LIN {X 0,Y 221.844,Z 433.494,A -85,B 0,C 180,E1 -25932.083,E2 -25932.083} C_VEL
LIN {X 0,Y 221.677,Z 433.43,A -85,B 0,C 180,E1 -25936.582,E2 -25936.582} C_VEL
LIN {X 0,Y 221.865,Z 433.946,A -85,B 0,C 180,E1 -25937.908,E2 -25937.908} C_VEL
LIN {X 0,Y 222.621,Z 436.665,A -85,B 0,C 180,E1 -25940.797,E2 -25940.797} C_VEL
LIN {X 0,Y 223.436,Z 440.266,A -85,B 0,C 180,E1 -25942.983,E2 -25942.983} C_VEL
LIN {X 0,Y 218.753,Z 475.978,A -85,B 0,C 180,E1 -25943.856,E2 -25943.856} C_VEL
LIN {X 0,Y 215.297,Z 491.744,A -85,B 0,C 180,E1 -25944.368,E2 -25944.368} C_VEL
LIN {X 0,Y 210.867,Z 506.328,A -85,B 0,C 180,E1 -25945.028,E2 -25945.028} C_VEL
LIN {X 0,Y 205.112,Z 520.999,A -85,B 0,C 180,E1 -25945.921,E2 -25945.921} C_VEL
LIN {X 0,Y 199.057,Z 533.652,A -85,B 0,C 180,E1 -25946.943,E2 -25946.943} C_VEL
LIN {X 0,Y 191.663,Z 546.67,A -85,B 0,C 180,E1 -25948.357,E2 -25948.357} C_VEL
LIN {X 0,Y 183.478,Z 558.958,A -85,B 0,C 180,E1 -25950.088,E2 -25950.088} C_VEL
LIN {X 0,Y 174.534,Z 570.553,A -85,B 0,C 180,E1 -25952.266,E2 -25952.266} C_VEL
LIN {X 0,Y 165.133,Z 581.209,A -85,B 0,C 180,E1 -25954.991,E2 -25954.991} C_VEL
LIN {X 0,Y 156.15,Z 590.141,A -85,B 0,C 180,E1 -25958.038,E2 -25958.038} C_VEL
LIN {X 0,Y 148.864,Z 596.686,A -85,B 0,C 180,E1 -25960.945,E2 -25960.945} C_VEL
LIN {X 0,Y 140.002,Z 603.992,A -85,B 0,C 180,E1 -25965.352,E2 -25965.352} C_VEL
LIN {X 0,Y 133.323,Z 608.926,A -85,B 0,C 180,E1 -25969.382,E2 -25969.382} C_VEL
LIN {X 0,Y 129.839,Z 611.007,A -85,B 0,C 180,E1 -25971.259,E2 -25971.259} C_VEL
LIN {X 0,Y 122.949,Z 614.076,A -85,B 0,C 180,E1 -25974.188,E2 -25974.188} C_VEL
LIN {X 0,Y 117.579,Z 616.128,A -85,B 0,C 180,E1 -25976.79,E2 -25976.79} C_VEL
LIN {X 0,Y 114.352,Z 617.413,A -85,B 0,C 180,E1 -25979.139,E2 -25979.139} C_VEL
LIN {X 0,Y 113.546,Z 617.817,A -85,B 0,C 180,E1 -25980.016,E2 -25980.016} C_VEL
LIN {X 0,Y 109.017,Z 620.077,A -85,B 0,C 180,E1 -25987.247,E2 -25987.247} C_VEL
LIN {X 0,Y 106.231,Z 621.156,A -85,B 0,C 180,E1 -25994.657,E2 -25994.657} C_VEL
LIN {X 0,Y 105.065,Z 621.173,A -85,B 0,C 180,E1 -26002.313,E2 -26002.313} C_VEL
LIN {X 0,Y 105.017,Z 620.759,A -85,B 0,C 180,E1 -26006.164,E2 -26006.164} C_VEL
LIN {X 0,Y 105.181,Z 620.031,A -85,B 0,C 180,E1 -26010.002,E2 -26010.002} C_VEL
LIN {X 0,Y 105.136,Z 617.616,A -85,B 0,C 180,E1 -26017.684,E2 -26017.684} C_VEL
LIN {X 0,Y 106.232,Z 613.919,A -85,B 0,C 180,E1 -26025.346,E2 -26025.346} C_VEL
LIN {X 0,Y 108.769,Z 608.839,A -85,B 0,C 180,E1 -26032.812,E2 -26032.812} C_VEL
LIN {X 0,Y 112.895,Z 602.246,A -85,B 0,C 180,E1 -26039.87,E2 -26039.87} C_VEL
LIN {X 0,Y 117.7,Z 595.095,A -85,B 0,C 180,E1 -26045.605,E2 -26045.605} C_VEL
LIN {X 0,Y 123.603,Z 586.461,A -85,B 0,C 180,E1 -26050.836,E2 -26050.836} C_VEL
LIN {X 0,Y 130.175,Z 576.16,A -85,B 0,C 180,E1 -26055.561,E2 -26055.561} C_VEL
LIN {X 0,Y 136.723,Z 565.278,A -85,B 0,C 180,E1 -26059.306,E2 -26059.306} C_VEL
LIN {X 0,Y 143.102,Z 553.613,A -85,B 0,C 180,E1 -26062.366,E2 -26062.366} C_VEL
LIN {X 0,Y 149.217,Z 540.906,A -85,B 0,C 180,E1 -26064.92,E2 -26064.92} C_VEL
LIN {X 0,Y 154.502,Z 528.264,A -85,B 0,C 180,E1 -26066.869,E2 -26066.869} C_VEL
LIN {X 0,Y 159.553,Z 513.659,A -85,B 0,C 180,E1 -26068.587,E2 -26068.587} C_VEL
LIN {X 0,Y 163.878,Z 498.558,A -85,B 0,C 180,E1 -26069.815,E2 -26069.815} C_VEL
LIN {X 0,Y 166.946,Z 483.72,A -85,B 0,C 180,E1 -26070.715,E2 -26070.715} C_VEL
LIN {X 0,Y 169.013,Z 467.946,A -85,B 0,C 180,E1 -26071.378,E2 -26071.378} C_VEL
LIN {X 0,Y 173.908,Z 418.093,A -85,B 0,C 180,E1 -26073.014,E2 -26073.014} C_VEL
LIN {X 0,Y 168.742,Z 404.265,A -85,B 0,C 180,E1 -26076.595,E2 -26076.595} C_VEL
LIN {X 0,Y 165.744,Z 397.177,A -85,B 0,C 180,E1 -26078.826,E2 -26078.826} C_VEL
LIN {X 0,Y 160.651,Z 388.212,A -85,B 0,C 180,E1 -26082.821,E2 -26082.821} C_VEL
LIN {X 0,Y 156.335,Z 381.165,A -85,B 0,C 180,E1 -26086.762,E2 -26086.762} C_VEL
LIN {X 0,Y 153.949,Z 377.355,A -85,B 0,C 180,E1 -26089.24,E2 -26089.24} C_VEL
LIN {X 0,Y 152.091,Z 374.461,A -85,B 0,C 180,E1 -26091.389,E2 -26091.389} C_VEL
LIN {X 0,Y 149.433,Z 370.221,A -85,B 0,C 180,E1 -26094.981,E2 -26094.981} C_VEL
LIN {X 0,Y 147.148,Z 366.725,A -85,B 0,C 180,E1 -26098.702,E2 -26098.702} C_VEL
LIN {X 0,Y 146.246,Z 365.497,A -85,B 0,C 180,E1 -26100.467,E2 -26100.467} C_VEL
LIN {X 0,Y 143.762,Z 361.234,A -85,B 0,C 180,E1 -26107.496,E2 -26107.496} C_VEL
LIN {X 0,Y 142.709,Z 361.006,A -85,B 0,C 180,E1 -26117.181,E2 -26117.181} C_VEL
LIN {X 0,Y 143.488,Z 361.557,A -85,B 0,C 180,E1 -26122.185,E2 -26122.185} C_VEL
LIN {X 0,Y 144.661,Z 364.587,A -85,B 0,C 180,E1 -26126.782,E2 -26126.782} C_VEL
LIN {X 0,Y 146.755,Z 366.776,A -85,B 0,C 180,E1 -26131.203,E2 -26131.203} C_VEL
LIN {X 0,Y 149.015,Z 370.336,A -85,B 0,C 180,E1 -26135.071,E2 -26135.071} C_VEL
LIN {X 0,Y 150.111,Z 371.757,A -85,B 0,C 180,E1 -26136.594,E2 -26136.594} C_VEL
LIN {X 0,Y 153.134,Z 376.335,A -85,B 0,C 180,E1 -26140.418,E2 -26140.418} C_VEL
LIN {X 0,Y 156.34,Z 381.231,A -85,B 0,C 180,E1 -26143.778,E2 -26143.778} C_VEL
LIN {X 0,Y 160.337,Z 387.689,A -85,B 0,C 180,E1 -26147.452,E2 -26147.452} C_VEL
LIN {X 0,Y 165.392,Z 396.474,A -85,B 0,C 180,E1 -26151.436,E2 -26151.436} C_VEL
LIN {X 0,Y 170.521,Z 406.407,A -85,B 0,C 180,E1 -26154.998,E2 -26154.998} C_VEL
LIN {X 0,Y 174.154,Z 413.847,A -85,B 0,C 180,E1 -26157.293,E2 -26157.293} C_VEL
LIN {X 0,Y 168.209,Z 471.305,A -85,B 0,C 180,E1 -26159.182,E2 -26159.182} C_VEL
LIN {X 0,Y 165.417,Z 487.206,A -85,B 0,C 180,E1 -26160.051,E2 -26160.051} C_VEL
LIN {X 0,Y 161.71,Z 502.382,A -85,B 0,C 180,E1 -26161.263,E2 -26161.263} C_VEL
LIN {X 0,Y 157.386,Z 516.243,A -85,B 0,C 180,E1 -26162.756,E2 -26162.756} C_VEL
LIN {X 0,Y 152.222,Z 529.97,A -85,B 0,C 180,E1 -26164.718,E2 -26164.718} C_VEL
LIN {X 0,Y 146.51,Z 542.733,A -85,B 0,C 180,E1 -26167.06,E2 -26167.06} C_VEL
LIN {X 0,Y 140.458,Z 554.57,A -85,B 0,C 180,E1 -26169.878,E2 -26169.878} C_VEL
LIN {X 0,Y 134.187,Z 565.53,A -85,B 0,C 180,E1 -26173.257,E2 -26173.257} C_VEL
LIN {X 0,Y 127.933,Z 575.611,A -85,B 0,C 180,E1 -26177.305,E2 -26177.305} C_VEL
LIN {X 0,Y 122.264,Z 584.145,A -85,B 0,C 180,E1 -26181.737,E2 -26181.737} C_VEL
LIN {X 0,Y 116.497,Z 592.511,A -85,B 0,C 180,E1 -26187.405,E2 -26187.405} C_VEL
LIN {X 0,Y 111.861,Z 599.37,A -85,B 0,C 180,E1 -26193.601,E2 -26193.601} C_VEL
LIN {X 0,Y 108.035,Z 605.6,A -85,B 0,C 180,E1 -26201.252,E2 -26201.252} C_VEL
LIN {X 0,Y 106.051,Z 609.293,A -85,B 0,C 180,E1 -26207.348,E2 -26207.348} C_VEL
LIN {X 0,Y 104.763,Z 612.126,A -85,B 0,C 180,E1 -26213.733,E2 -26213.733} C_VEL
LIN {X 0,Y 104.422,Z 613.834,A -85,B 0,C 180,E1 -26218.976,E2 -26218.976} C_VEL
LIN {X 0,Y 104.917,Z 615.375,A -85,B 0,C 180,E1 -26227.073,E2 -26227.073} C_VEL
LIN {X 0,Y 106.415,Z 615.735,A -85,B 0,C 180,E1 -26233.418,E2 -26233.418} C_VEL
LIN {X 0,Y 109.255,Z 615.219,A -85,B 0,C 180,E1 -26240.522,E2 -26240.522} C_VEL
LIN {X 0,Y 112.414,Z 614.078,A -85,B 0,C 180,E1 -26245.767,E2 -26245.767} C_VEL
LIN {X 0,Y 118.398,Z 611.322,A -85,B 0,C 180,E1 -26252.916,E2 -26252.916} C_VEL
LIN {X 0,Y 124.722,Z 607.892,A -85,B 0,C 180,E1 -26258.391,E2 -26258.391} C_VEL
LIN {X 0,Y 132.053,Z 603.355,A -85,B 0,C 180,E1 -26263.323,E2 -26263.323} C_VEL
LIN {X 0,Y 139.8,Z 598.023,A -85,B 0,C 180,E1 -26267.477,E2 -26267.477} C_VEL
LIN {X 0,Y 149.217,Z 590.776,A -85,B 0,C 180,E1 -26271.511,E2 -26271.511} C_VEL
LIN {X 0,Y 158.751,Z 582.367,A -85,B 0,C 180,E1 -26274.925,E2 -26274.925} C_VEL
LIN {X 0,Y 167.666,Z 573.428,A -85,B 0,C 180,E1 -26277.602,E2 -26277.602} C_VEL
LIN {X 0,Y 176.942,Z 562.763,A -85,B 0,C 180,E1 -26280.004,E2 -26280.004} C_VEL
LIN {X 0,Y 185.165,Z 551.838,A -85,B 0,C 180,E1 -26281.903,E2 -26281.903} C_VEL
LIN {X 0,Y 192.726,Z 540.213,A -85,B 0,C 180,E1 -26283.456,E2 -26283.456} C_VEL
LIN {X 0,Y 200.122,Z 526.794,A -85,B 0,C 180,E1 -26284.826,E2 -26284.826} C_VEL
LIN {X 0,Y 206.121,Z 513.569,A -85,B 0,C 180,E1 -26285.874,E2 -26285.874} C_VEL
LIN {X 0,Y 211.446,Z 498.933,A -85,B 0,C 180,E1 -26286.754,E2 -26286.754} C_VEL
LIN {X 0,Y 215.645,Z 483.814,A -85,B 0,C 180,E1 -26287.396,E2 -26287.396} C_VEL
LIN {X 0,Y 218.573,Z 468.573,A -85,B 0,C 180,E1 -26287.838,E2 -26287.838} C_VEL
LIN {X 0,Y 221.846,Z 443.6,A -85,B 0,C 180,E1 -26288.43,E2 -26288.43} C_VEL
LIN {X 0,Y 220.843,Z 440.514,A -85,B 0,C 180,E1 -26292.175,E2 -26292.175} C_VEL
LIN {X 0,Y 220.703,Z 440.483,A -85,B 0,C 180,E1 -26296.657,E2 -26296.657} C_VEL
LIN {X 0,Y 220.854,Z 441.063,A -85,B 0,C 180,E1 -26297.845,E2 -26297.845} C_VEL
LIN {X 0,Y 221.442,Z 443.47,A -85,B 0,C 180,E1 -26300.346,E2 -26300.346} C_VEL
LIN {X 0,Y 221.716,Z 444.897,A -85,B 0,C 180,E1 -26301.284,E2 -26301.284} C_VEL
LIN {X 0,Y 217.512,Z 475.713,A -85,B 0,C 180,E1 -26302.01,E2 -26302.01} C_VEL
LIN {X 0,Y 214.065,Z 491.149,A -85,B 0,C 180,E1 -26302.483,E2 -26302.483} C_VEL
LIN {X 0,Y 209.628,Z 505.616,A -85,B 0,C 180,E1 -26303.098,E2 -26303.098} C_VEL
LIN {X 0,Y 203.737,Z 520.418,A -85,B 0,C 180,E1 -26303.922,E2 -26303.922} C_VEL
LIN {X 0,Y 196.788,Z 534.515,A -85,B 0,C 180,E1 -26305.015,E2 -26305.015} C_VEL
LIN {X 0,Y 189.223,Z 547.349,A -85,B 0,C 180,E1 -26306.363,E2 -26306.363} C_VEL
LIN {X 0,Y 180.87,Z 559.394,A -85,B 0,C 180,E1 -26308.007,E2 -26308.007} C_VEL
LIN {X 0,Y 172.361,Z 570.035,A -85,B 0,C 180,E1 -26309.954,E2 -26309.954} C_VEL
LIN {X 0,Y 162.588,Z 580.754,A -85,B 0,C 180,E1 -26312.556,E2 -26312.556} C_VEL
LIN {X 0,Y 154.534,Z 588.515,A -85,B 0,C 180,E1 -26315.057,E2 -26315.057} C_VEL
LIN {X 0,Y 144.322,Z 597.263,A -85,B 0,C 180,E1 -26318.821,E2 -26318.821} C_VEL
LIN {X 0,Y 135.022,Z 604.398,A -85,B 0,C 180,E1 -26323.225,E2 -26323.225} C_VEL
LIN {X 0,Y 126.569,Z 610.15,A -85,B 0,C 180,E1 -26328.219,E2 -26328.219} C_VEL
LIN {X 0,Y 119.315,Z 614.638,A -85,B 0,C 180,E1 -26333.915,E2 -26333.915} C_VEL
LIN {X 0,Y 113.546,Z 617.817,A -85,B 0,C 180,E1 -26340.016,E2 -26340.016} C_VEL
LIN {X 0,Y 110.899,Z 618.907,A -85,B 0,C 180,E1 -26342.656,E2 -26342.656} C_VEL
LIN {X 0,Y 105.402,Z 620.175,A -85,B 0,C 180,E1 -26346.98,E2 -26346.98} C_VEL
LIN {X 0,Y 101.336,Z 620.779,A -85,B 0,C 180,E1 -26350.759,E2 -26350.759} C_VEL
LIN {X 0,Y 99.317,Z 621,A -85,B 0,C 180,E1 -26353.938,E2 -26353.938} C_VEL
LIN {X 0,Y 98.964,Z 621.01,A -85,B 0,C 180,E1 -26355.06,E2 -26355.06} C_VEL
LIN {X 0,Y 98.017,Z 620.882,A -85,B 0,C 180,E1 -26361.757,E2 -26361.757} C_VEL
LIN {X 0,Y 98.084,Z 619.681,A -85,B 0,C 180,E1 -26370.002,E2 -26370.002} C_VEL
LIN {X 0,Y 98.073,Z 617.166,A -85,B 0,C 180,E1 -26378.242,E2 -26378.242} C_VEL
LIN {X 0,Y 99.347,Z 613.356,A -85,B 0,C 180,E1 -26386.439,E2 -26386.439} C_VEL
LIN {X 0,Y 102.176,Z 608.154,A -85,B 0,C 180,E1 -26394.376,E2 -26394.376} C_VEL
LIN {X 0,Y 106.729,Z 601.436,A -85,B 0,C 180,E1 -26401.79,E2 -26401.79} C_VEL
LIN {X 0,Y 111.921,Z 594.141,A -85,B 0,C 180,E1 -26407.753,E2 -26407.753} C_VEL
LIN {X 0,Y 118.225,Z 585.346,A -85,B 0,C 180,E1 -26413.129,E2 -26413.129} C_VEL
LIN {X 0,Y 124.257,Z 576.36,A -85,B 0,C 180,E1 -26417.332,E2 -26417.332} C_VEL
LIN {X 0,Y 130.974,Z 565.762,A -85,B 0,C 180,E1 -26421.084,E2 -26421.084} C_VEL
LIN {X 0,Y 137.569,Z 554.227,A -85,B 0,C 180,E1 -26424.195,E2 -26424.195} C_VEL
LIN {X 0,Y 143.876,Z 541.681,A -85,B 0,C 180,E1 -26426.774,E2 -26426.774} C_VEL
LIN {X 0,Y 149.164,Z 529.55,A -85,B 0,C 180,E1 -26428.674,E2 -26428.674} C_VEL
LIN {X 0,Y 154.547,Z 514.901,A -85,B 0,C 180,E1 -26430.424,E2 -26430.424} C_VEL
LIN {X 0,Y 159.139,Z 499.606,A -85,B 0,C 180,E1 -26431.702,E2 -26431.702} C_VEL
LIN {X 0,Y 162.481,Z 484.298,A -85,B 0,C 180,E1 -26432.631,E2 -26432.631} C_VEL
LIN {X 0,Y 164.699,Z 468.218,A -85,B 0,C 180,E1 -26433.309,E2 -26433.309} C_VEL
LIN {X 0,Y 169.582,Z 420.714,A -85,B 0,C 180,E1 -26434.829,E2 -26434.829} C_VEL
LIN {X 0,Y 164.978,Z 408.11,A -85,B 0,C 180,E1 -26438.259,E2 -26438.259} C_VEL
LIN {X 0,Y 162.603,Z 402.275,A -85,B 0,C 180,E1 -26440.185,E2 -26440.185} C_VEL
LIN {X 0,Y 157.88,Z 393.684,A -85,B 0,C 180,E1 -26444.132,E2 -26444.132} C_VEL
LIN {X 0,Y 154.164,Z 387.35,A -85,B 0,C 180,E1 -26447.768,E2 -26447.768} C_VEL
LIN {X 0,Y 150.644,Z 381.382,A -85,B 0,C 180,E1 -26451.821,E2 -26451.821} C_VEL
LIN {X 0,Y 147.643,Z 376.643,A -85,B 0,C 180,E1 -26456.035,E2 -26456.035} C_VEL
LIN {X 0,Y 145.236,Z 372.637,A -85,B 0,C 180,E1 -26460.47,E2 -26460.47} C_VEL
LIN {X 0,Y 142.641,Z 368.229,A -85,B 0,C 180,E1 -26468.025,E2 -26468.025} C_VEL
LIN {X 0,Y 141.739,Z 368.046,A -85,B 0,C 180,E1 -26477.303,E2 -26477.303} C_VEL
LIN {X 0,Y 142.382,Z 368.528,A -85,B 0,C 180,E1 -26481.694,E2 -26481.694} C_VEL
LIN {X 0,Y 143.544,Z 371.549,A -85,B 0,C 180,E1 -26486.464,E2 -26486.464} C_VEL
LIN {X 0,Y 145.365,Z 373.52,A -85,B 0,C 180,E1 -26490.485,E2 -26490.485} C_VEL
LIN {X 0,Y 147.667,Z 377.231,A -85,B 0,C 180,E1 -26494.638,E2 -26494.638} C_VEL
LIN {X 0,Y 151.024,Z 382.367,A -85,B 0,C 180,E1 -26499.246,E2 -26499.246} C_VEL
LIN {X 0,Y 154.084,Z 387.287,A -85,B 0,C 180,E1 -26502.701,E2 -26502.701} C_VEL
LIN {X 0,Y 157.928,Z 393.777,A -85,B 0,C 180,E1 -26506.443,E2 -26506.443} C_VEL
LIN {X 0,Y 162.445,Z 401.904,A -85,B 0,C 180,E1 -26510.209,E2 -26510.209} C_VEL
LIN {X 0,Y 167.373,Z 411.835,A -85,B 0,C 180,E1 -26513.875,E2 -26513.875} C_VEL
LIN {X 0,Y 169.693,Z 416.598,A -85,B 0,C 180,E1 -26515.426,E2 -26515.426} C_VEL
LIN {X 0,Y 164,Z 470.802,A -85,B 0,C 180,E1 -26517.215,E2 -26517.215} C_VEL
LIN {X 0,Y 161.188,Z 486.591,A -85,B 0,C 180,E1 -26518.045,E2 -26518.045} C_VEL
LIN {X 0,Y 157.316,Z 502.181,A -85,B 0,C 180,E1 -26519.271,E2 -26519.271} C_VEL
LIN {X 0,Y 152.841,Z 516.114,A -85,B 0,C 180,E1 -26520.744,E2 -26520.744} C_VEL
LIN {X 0,Y 147.472,Z 529.928,A -85,B 0,C 180,E1 -26522.697,E2 -26522.697} C_VEL
LIN {X 0,Y 141.564,Z 542.72,A -85,B 0,C 180,E1 -26525.039,E2 -26525.039} C_VEL
LIN {X 0,Y 135.052,Z 554.946,A -85,B 0,C 180,E1 -26527.964,E2 -26527.964} C_VEL
LIN {X 0,Y 128.135,Z 566.506,A -85,B 0,C 180,E1 -26531.615,E2 -26531.615} C_VEL
LIN {X 0,Y 121.733,Z 576.331,A -85,B 0,C 180,E1 -26535.723,E2 -26535.723} C_VEL
LIN {X 0,Y 114.807,Z 586.182,A -85,B 0,C 180,E1 -26541.174,E2 -26541.174} C_VEL
LIN {X 0,Y 108.942,Z 594.247,A -85,B 0,C 180,E1 -26547.225,E2 -26547.225} C_VEL
LIN {X 0,Y 104.264,Z 600.812,A -85,B 0,C 180,E1 -26553.863,E2 -26553.863} C_VEL
LIN {X 0,Y 100.458,Z 606.774,A -85,B 0,C 180,E1 -26562.113,E2 -26562.113} C_VEL
LIN {X 0,Y 98.525,Z 610.215,A -85,B 0,C 180,E1 -26568.721,E2 -26568.721} C_VEL
LIN {X 0,Y 97.441,Z 612.917,A -85,B 0,C 180,E1 -26575.64,E2 -26575.64} C_VEL
LIN {X 0,Y 97.314,Z 614.232,A -85,B 0,C 180,E1 -26580.364,E2 -26580.364} C_VEL
LIN {X 0,Y 97.911,Z 615.531,A -85,B 0,C 180,E1 -26587.867,E2 -26587.867} C_VEL
LIN {X 0,Y 99.781,Z 615.947,A -85,B 0,C 180,E1 -26595.234,E2 -26595.234} C_VEL
LIN {X 0,Y 103.924,Z 615.152,A -85,B 0,C 180,E1 -26604.24,E2 -26604.24} C_VEL
LIN {X 0,Y 106.968,Z 614.139,A -85,B 0,C 180,E1 -26608.658,E2 -26608.658} C_VEL
LIN {X 0,Y 111.409,Z 612.324,A -85,B 0,C 180,E1 -26613.803,E2 -26613.803} C_VEL
LIN {X 0,Y 119.269,Z 608.494,A -85,B 0,C 180,E1 -26620.521,E2 -26620.521} C_VEL
LIN {X 0,Y 127.019,Z 604.108,A -85,B 0,C 180,E1 -26625.521,E2 -26625.521} C_VEL
LIN {X 0,Y 137.2,Z 597.513,A -85,B 0,C 180,E1 -26630.598,E2 -26630.598} C_VEL
LIN {X 0,Y 147.256,Z 590.006,A -85,B 0,C 180,E1 -26634.527,E2 -26634.527} C_VEL
LIN {X 0,Y 156.99,Z 581.655,A -85,B 0,C 180,E1 -26637.688,E2 -26637.688} C_VEL
LIN {X 0,Y 166.65,Z 572.198,A -85,B 0,C 180,E1 -26640.331,E2 -26640.331} C_VEL
LIN {X 0,Y 175.86,Z 561.812,A -85,B 0,C 180,E1 -26642.498,E2 -26642.498} C_VEL
LIN {X 0,Y 184.832,Z 550.011,A -85,B 0,C 180,E1 -26644.365,E2 -26644.365} C_VEL
LIN {X 0,Y 193.313,Z 536.828,A -85,B 0,C 180,E1 -26645.93,E2 -26645.93} C_VEL
LIN {X 0,Y 200.533,Z 523.42,A -85,B 0,C 180,E1 -26647.152,E2 -26647.152} C_VEL
LIN {X 0,Y 206.76,Z 509.222,A -85,B 0,C 180,E1 -26648.128,E2 -26648.128} C_VEL
LIN {X 0,Y 211.947,Z 494.116,A -85,B 0,C 180,E1 -26648.883,E2 -26648.883} C_VEL
LIN {X 0,Y 215.763,Z 479.081,A -85,B 0,C 180,E1 -26649.415,E2 -26649.415} C_VEL
LIN {X 0,Y 218.518,Z 462.45,A -85,B 0,C 180,E1 -26649.829,E2 -26649.829} C_VEL
LIN {X 0,Y 220.215,Z 449.373,A -85,B 0,C 180,E1 -26650.158,E2 -26650.158} C_VEL
LIN {X 0,Y 219.793,Z 447.439,A -85,B 0,C 180,E1 -26652.585,E2 -26652.585} C_VEL
LIN {X 0,Y 219.774,Z 447.598,A -85,B 0,C 180,E1 -26657.045,E2 -26657.045} C_VEL
LIN {X 0,Y 220.206,Z 449.797,A -85,B 0,C 180,E1 -26659.567,E2 -26659.567} C_VEL
LIN {X 0,Y 216.488,Z 475.973,A -85,B 0,C 180,E1 -26660.156,E2 -26660.156} C_VEL
LIN {X 0,Y 212.898,Z 491.554,A -85,B 0,C 180,E1 -26660.606,E2 -26660.606} C_VEL
LIN {X 0,Y 208.228,Z 506.217,A -85,B 0,C 180,E1 -26661.196,E2 -26661.196} C_VEL
LIN {X 0,Y 202.638,Z 519.938,A -85,B 0,C 180,E1 -26661.917,E2 -26661.917} C_VEL
LIN {X 0,Y 195.515,Z 534.05,A -85,B 0,C 180,E1 -26662.915,E2 -26662.915} C_VEL
LIN {X 0,Y 187.014,Z 548.026,A -85,B 0,C 180,E1 -26664.317,E2 -26664.317} C_VEL
LIN {X 0,Y 177.836,Z 560.711,A -85,B 0,C 180,E1 -26665.996,E2 -26665.996} C_VEL
LIN {X 0,Y 168.977,Z 571.298,A -85,B 0,C 180,E1 -26667.898,E2 -26667.898} C_VEL
LIN {X 0,Y 160.338,Z 580.338,A -85,B 0,C 180,E1 -26670.042,E2 -26670.042} C_VEL
LIN {X 0,Y 150.596,Z 589.311,A -85,B 0,C 180,E1 -26672.862,E2 -26672.862} C_VEL
LIN {X 0,Y 142.573,Z 595.901,A -85,B 0,C 180,E1 -26675.579,E2 -26675.579} C_VEL
LIN {X 0,Y 133.341,Z 602.734,A -85,B 0,C 180,E1 -26679.398,E2 -26679.398} C_VEL
LIN {X 0,Y 123.513,Z 609.176,A -85,B 0,C 180,E1 -26684.665,E2 -26684.665} C_VEL
LIN {X 0,Y 115.431,Z 613.814,A -85,B 0,C 180,E1 -26690.264,E2 -26690.264} C_VEL
LIN {X 0,Y 107.21,Z 617.976,A -85,B 0,C 180,E1 -26698.373,E2 -26698.373} C_VEL
LIN {X 0,Y 102.438,Z 620.013,A -85,B 0,C 180,E1 -26705.694,E2 -26705.694} C_VEL
LIN {X 0,Y 98.964,Z 621.01,A -85,B 0,C 180,E1 -26715.06,E2 -26715.06} C_VEL
LIN {X 0,Y 97.699,Z 621.037,A -85,B 0,C 180,E1 -26718.421,E2 -26718.421} C_VEL
LIN {X 0,Y 95.789,Z 620.797,A -85,B 0,C 180,E1 -26721.75,E2 -26721.75} C_VEL
LIN {X 0,Y 91.907,Z 619.619,A -85,B 0,C 180,E1 -26728.663,E2 -26728.663} C_VEL
LIN {X 0,Y 90.845,Z 618.369,A -85,B 0,C 180,E1 -26733.589,E2 -26733.589} C_VEL
LIN {X 0,Y 91.035,Z 616.698,A -85,B 0,C 180,E1 -26738.884,E2 -26738.884} C_VEL
LIN {X 0,Y 92.483,Z 612.769,A -85,B 0,C 180,E1 -26747.698,E2 -26747.698} C_VEL
LIN {X 0,Y 95.674,Z 607.436,A -85,B 0,C 180,E1 -26756.153,E2 -26756.153} C_VEL
LIN {X 0,Y 100.676,Z 600.577,A -85,B 0,C 180,E1 -26763.951,E2 -26763.951} C_VEL
LIN {X 0,Y 106.325,Z 593.132,A -85,B 0,C 180,E1 -26770.127,E2 -26770.127} C_VEL
LIN {X 0,Y 112.063,Z 585.551,A -85,B 0,C 180,E1 -26774.874,E2 -26774.874} C_VEL
LIN {X 0,Y 119.486,Z 574.977,A -85,B 0,C 180,E1 -26779.876,E2 -26779.876} C_VEL
LIN {X 0,Y 126.562,Z 564.146,A -85,B 0,C 180,E1 -26783.629,E2 -26783.629} C_VEL
LIN {X 0,Y 133.497,Z 552.339,A -85,B 0,C 180,E1 -26786.694,E2 -26786.694} C_VEL
LIN {X 0,Y 140.092,Z 539.454,A -85,B 0,C 180,E1 -26789.217,E2 -26789.217} C_VEL
LIN {X 0,Y 146.103,Z 525.65,A -85,B 0,C 180,E1 -26791.243,E2 -26791.243} C_VEL
LIN {X 0,Y 151.135,Z 511.629,A -85,B 0,C 180,E1 -26792.79,E2 -26792.79} C_VEL
LIN {X 0,Y 155.502,Z 496.728,A -85,B 0,C 180,E1 -26793.93,E2 -26793.93} C_VEL
LIN {X 0,Y 158.572,Z 482.351,A -85,B 0,C 180,E1 -26794.745,E2 -26794.745} C_VEL
LIN {X 0,Y 160.837,Z 465.264,A -85,B 0,C 180,E1 -26795.426,E2 -26795.426} C_VEL
LIN {X 0,Y 165.27,Z 423.126,A -85,B 0,C 180,E1 -26796.771,E2 -26796.771} C_VEL
LIN {X 0,Y 160.796,Z 410.229,A -85,B 0,C 180,E1 -26800.516,E2 -26800.516} C_VEL
LIN {X 0,Y 158.598,Z 405.594,A -85,B 0,C 180,E1 -26802.363,E2 -26802.363} C_VEL
LIN {X 0,Y 154.664,Z 398.121,A -85,B 0,C 180,E1 -26806.027,E2 -26806.027} C_VEL
LIN {X 0,Y 150.134,Z 390.177,A -85,B 0,C 180,E1 -26811.016,E2 -26811.016} C_VEL
LIN {X 0,Y 148.158,Z 386.858,A -85,B 0,C 180,E1 -26813.659,E2 -26813.659} C_VEL
LIN {X 0,Y 145.92,Z 383.059,A -85,B 0,C 180,E1 -26817.097,E2 -26817.097} C_VEL
LIN {X 0,Y 143.885,Z 379.379,A -85,B 0,C 180,E1 -26821.184,E2 -26821.184} C_VEL
LIN {X 0,Y 141.534,Z 375.197,A -85,B 0,C 180,E1 -26828.562,E2 -26828.562} C_VEL
LIN {X 0,Y 140.868,Z 375.162,A -85,B 0,C 180,E1 -26838.573,E2 -26838.573} C_VEL
LIN {X 0,Y 141.303,Z 375.607,A -85,B 0,C 180,E1 -26841.329,E2 -26841.329} C_VEL
LIN {X 0,Y 142.501,Z 378.617,A -85,B 0,C 180,E1 -26846.345,E2 -26846.345} C_VEL
LIN {X 0,Y 143.982,Z 380.292,A -85,B 0,C 180,E1 -26849.764,E2 -26849.764} C_VEL
LIN {X 0,Y 146.35,Z 384.158,A -85,B 0,C 180,E1 -26854.236,E2 -26854.236} C_VEL
LIN {X 0,Y 149.476,Z 389.343,A -85,B 0,C 180,E1 -26858.72,E2 -26858.72} C_VEL
LIN {X 0,Y 152.907,Z 395.012,A -85,B 0,C 180,E1 -26862.7,E2 -26862.7} C_VEL
LIN {X 0,Y 157.049,Z 402.59,A -85,B 0,C 180,E1 -26866.792,E2 -26866.792} C_VEL
LIN {X 0,Y 161.414,Z 411.162,A -85,B 0,C 180,E1 -26870.483,E2 -26870.483} C_VEL
LIN {X 0,Y 165.451,Z 419.732,A -85,B 0,C 180,E1 -26873.554,E2 -26873.554} C_VEL
LIN {X 0,Y 159.747,Z 471.415,A -85,B 0,C 180,E1 -26875.211,E2 -26875.211} C_VEL
LIN {X 0,Y 156.836,Z 487.13,A -85,B 0,C 180,E1 -26876.031,E2 -26876.031} C_VEL
LIN {X 0,Y 153.089,Z 501.817,A -85,B 0,C 180,E1 -26877.16,E2 -26877.16} C_VEL
LIN {X 0,Y 148.463,Z 515.901,A -85,B 0,C 180,E1 -26878.619,E2 -26878.619} C_VEL
LIN {X 0,Y 142.925,Z 529.754,A -85,B 0,C 180,E1 -26880.545,E2 -26880.545} C_VEL
LIN {X 0,Y 136.135,Z 543.854,A -85,B 0,C 180,E1 -26883.145,E2 -26883.145} C_VEL
LIN {X 0,Y 129.174,Z 556.313,A -85,B 0,C 180,E1 -26886.215,E2 -26886.215} C_VEL
LIN {X 0,Y 122.208,Z 567.364,A -85,B 0,C 180,E1 -26889.814,E2 -26889.814} C_VEL
LIN {X 0,Y 115.438,Z 577.247,A -85,B 0,C 180,E1 -26894.099,E2 -26894.099} C_VEL
LIN {X 0,Y 109.243,Z 585.596,A -85,B 0,C 180,E1 -26898.871,E2 -26898.871} C_VEL
LIN {X 0,Y 102.941,Z 593.776,A -85,B 0,C 180,E1 -26905.103,E2 -26905.103} C_VEL
LIN {X 0,Y 97.603,Z 600.815,A -85,B 0,C 180,E1 -26912.462,E2 -26912.462} C_VEL
LIN {X 0,Y 94.558,Z 605.183,A -85,B 0,C 180,E1 -26918.547,E2 -26918.547} C_VEL
LIN {X 0,Y 92.201,Z 609.023,A -85,B 0,C 180,E1 -26925.471,E2 -26925.471} C_VEL
LIN {X 0,Y 90.623,Z 612.038,A -85,B 0,C 180,E1 -26932.813,E2 -26932.813} C_VEL
LIN {X 0,Y 90.223,Z 614.416,A -85,B 0,C 180,E1 -26941.051,E2 -26941.051} C_VEL
LIN {X 0,Y 91.09,Z 615.773,A -85,B 0,C 180,E1 -26949.52,E2 -26949.52} C_VEL
LIN {X 0,Y 93.73,Z 616.134,A -85,B 0,C 180,E1 -26958.57,E2 -26958.57} C_VEL
LIN {X 0,Y 96.543,Z 615.72,A -85,B 0,C 180,E1 -26964.392,E2 -26964.392} C_VEL
LIN {X 0,Y 102.664,Z 613.918,A -85,B 0,C 180,E1 -26972.859,E2 -26972.859} C_VEL
LIN {X 0,Y 109.071,Z 611.368,A -85,B 0,C 180,E1 -26979.109,E2 -26979.109} C_VEL
LIN {X 0,Y 116.617,Z 607.858,A -85,B 0,C 180,E1 -26984.624,E2 -26984.624} C_VEL
LIN {X 0,Y 127.277,Z 601.952,A -85,B 0,C 180,E1 -26990.47,E2 -26990.47} C_VEL
LIN {X 0,Y 138.001,Z 594.993,A -85,B 0,C 180,E1 -26994.942,E2 -26994.942} C_VEL
LIN {X 0,Y 147.653,Z 587.8,A -85,B 0,C 180,E1 -26998.216,E2 -26998.216} C_VEL
LIN {X 0,Y 158.156,Z 578.76,A -85,B 0,C 180,E1 -27001.167,E2 -27001.167} C_VEL
LIN {X 0,Y 167.426,Z 569.522,A -85,B 0,C 180,E1 -27003.392,E2 -27003.392} C_VEL
LIN {X 0,Y 177.376,Z 558.1,A -85,B 0,C 180,E1 -27005.457,E2 -27005.457} C_VEL
LIN {X 0,Y 185.857,Z 546.728,A -85,B 0,C 180,E1 -27006.984,E2 -27006.984} C_VEL
LIN {X 0,Y 192.964,Z 535.614,A -85,B 0,C 180,E1 -27008.163,E2 -27008.163} C_VEL
LIN {X 0,Y 200.056,Z 522.465,A -85,B 0,C 180,E1 -27009.261,E2 -27009.261} C_VEL
LIN {X 0,Y 206.062,Z 508.859,A -85,B 0,C 180,E1 -27010.115,E2 -27010.115} C_VEL
LIN {X 0,Y 211.295,Z 493.743,A -85,B 0,C 180,E1 -27010.82,E2 -27010.82} C_VEL
LIN {X 0,Y 215.154,Z 478.682,A -85,B 0,C 180,E1 -27011.305,E2 -27011.305} C_VEL
LIN {X 0,Y 217.898,Z 462.347,A -85,B 0,C 180,E1 -27011.692,E2 -27011.692} C_VEL
LIN {X 0,Y 218.869,Z 455.137,A -85,B 0,C 180,E1 -27011.852,E2 -27011.852} C_VEL
LIN {X 0,Y 218.752,Z 454.388,A -85,B 0,C 180,E1 -27012.999,E2 -27012.999} C_VEL
LIN {X 0,Y 218.76,Z 454.7,A -85,B 0,C 180,E1 -27016.93,E2 -27016.93} C_VEL
LIN {X 0,Y 218.829,Z 455.509,A -85,B 0,C 180,E1 -27017.828,E2 -27017.828} C_VEL
LIN {X 0,Y 215.533,Z 477.127,A -85,B 0,C 180,E1 -27018.313,E2 -27018.313} C_VEL
LIN {X 0,Y 211.521,Z 493.48,A -85,B 0,C 180,E1 -27018.763,E2 -27018.763} C_VEL
LIN {X 0,Y 206.254,Z 508.992,A -85,B 0,C 180,E1 -27019.369,E2 -27019.369} C_VEL
LIN {X 0,Y 200.176,Z 522.926,A -85,B 0,C 180,E1 -27020.094,E2 -27020.094} C_VEL
LIN {X 0,Y 193.736,Z 535.086,A -85,B 0,C 180,E1 -27020.92,E2 -27020.92} C_VEL
LIN {X 0,Y 185.838,Z 547.695,A -85,B 0,C 180,E1 -27022.104,E2 -27022.104} C_VEL
LIN {X 0,Y 176.48,Z 560.297,A -85,B 0,C 180,E1 -27023.667,E2 -27023.667} C_VEL
LIN {X 0,Y 167.335,Z 570.926,A -85,B 0,C 180,E1 -27025.451,E2 -27025.451} C_VEL
LIN {X 0,Y 156.941,Z 581.384,A -85,B 0,C 180,E1 -27027.824,E2 -27027.824} C_VEL
LIN {X 0,Y 146.894,Z 590.169,A -85,B 0,C 180,E1 -27030.553,E2 -27030.553} C_VEL
LIN {X 0,Y 135.897,Z 598.505,A -85,B 0,C 180,E1 -27034.167,E2 -27034.167} C_VEL
LIN {X 0,Y 125.704,Z 605.294,A -85,B 0,C 180,E1 -27038.493,E2 -27038.493} C_VEL
LIN {X 0,Y 116.324,Z 610.72,A -85,B 0,C 180,E1 -27043.534,E2 -27043.534} C_VEL
LIN {X 0,Y 108.091,Z 614.915,A -85,B 0,C 180,E1 -27049.447,E2 -27049.447} C_VEL
LIN {X 0,Y 100.459,Z 618.258,A -85,B 0,C 180,E1 -27057.098,E2 -27057.098} C_VEL
LIN {X 0,Y 95.947,Z 619.959,A -85,B 0,C 180,E1 -27063.931,E2 -27063.931} C_VEL
LIN {X 0,Y 92.488,Z 620.8,A -85,B 0,C 180,E1 -27072.307,E2 -27072.307} C_VEL
LIN {X 0,Y 90.963,Z 620.592,A -85,B 0,C 180,E1 -27081.113,E2 -27081.113} C_VEL
LIN {X 0,Y 90.848,Z 620.081,A -85,B 0,C 180,E1 -27085.565,E2 -27085.565} C_VEL
LIN {X 0,Y 90.982,Z 619.282,A -85,B 0,C 180,E1 -27090.002,E2 -27090.002} C_VEL
LIN {X 0,Y 90.845,Z 618.369,A -85,B 0,C 180,E1 -27093.589,E2 -27093.589} C_VEL
LIN {X 0,Y 90.596,Z 617.669,A -85,B 0,C 180,E1 -27096.026,E2 -27096.026} C_VEL
LIN {X 0,Y 89.497,Z 616.385,A -85,B 0,C 180,E1 -27099.639,E2 -27099.639} C_VEL
LIN {X 0,Y 86.624,Z 612.605,A -85,B 0,C 180,E1 -27108.203,E2 -27108.203} C_VEL
LIN {X 0,Y 86.68,Z 610.636,A -85,B 0,C 180,E1 -27111.944,E2 -27111.944} C_VEL
LIN {X 0,Y 87.035,Z 609.959,A -85,B 0,C 180,E1 -27113.16,E2 -27113.16} C_VEL
LIN {X 0,Y 90.497,Z 605.073,A -85,B 0,C 180,E1 -27120.319,E2 -27120.319} C_VEL
LIN {X 0,Y 96.399,Z 597.642,A -85,B 0,C 180,E1 -27128.295,E2 -27128.295} C_VEL
LIN {X 0,Y 102.957,Z 589.665,A -85,B 0,C 180,E1 -27134.402,E2 -27134.402} C_VEL
LIN {X 0,Y 110.308,Z 579.986,A -85,B 0,C 180,E1 -27139.867,E2 -27139.867} C_VEL
LIN {X 0,Y 117.418,Z 570.129,A -85,B 0,C 180,E1 -27143.905,E2 -27143.905} C_VEL
LIN {X 0,Y 125.026,Z 558.39,A -85,B 0,C 180,E1 -27147.478,E2 -27147.478} C_VEL
LIN {X 0,Y 131.715,Z 546.76,A -85,B 0,C 180,E1 -27150.119,E2 -27150.119} C_VEL
LIN {X 0,Y 137.958,Z 534.322,A -85,B 0,C 180,E1 -27152.251,E2 -27152.251} C_VEL
LIN {X 0,Y 143.422,Z 521.326,A -85,B 0,C 180,E1 -27153.971,E2 -27153.971} C_VEL
LIN {X 0,Y 148.382,Z 507.155,A -85,B 0,C 180,E1 -27155.34,E2 -27155.34} C_VEL
LIN {X 0,Y 152.431,Z 492.215,A -85,B 0,C 180,E1 -27156.399,E2 -27156.399} C_VEL
LIN {X 0,Y 155.351,Z 477.472,A -85,B 0,C 180,E1 -27157.097,E2 -27157.097} C_VEL
LIN {X 0,Y 159.595,Z 440.466,A -85,B 0,C 180,E1 -27158.317,E2 -27158.317} C_VEL
LIN {X 0,Y 161.197,Z 425.716,A -85,B 0,C 180,E1 -27158.778,E2 -27158.778} C_VEL
LIN {X 0,Y 157.345,Z 414.298,A -85,B 0,C 180,E1 -27162.281,E2 -27162.281} C_VEL
LIN {X 0,Y 153.399,Z 406.183,A -85,B 0,C 180,E1 -27166.05,E2 -27166.05} C_VEL
LIN {X 0,Y 149.661,Z 399.26,A -85,B 0,C 180,E1 -27170.156,E2 -27170.156} C_VEL
LIN {X 0,Y 146.856,Z 394.003,A -85,B 0,C 180,E1 -27173.942,E2 -27173.942} C_VEL
LIN {X 0,Y 144.334,Z 389.591,A -85,B 0,C 180,E1 -27178.015,E2 -27178.015} C_VEL
LIN {X 0,Y 142.537,Z 386.118,A -85,B 0,C 180,E1 -27181.892,E2 -27181.892} C_VEL
LIN {X 0,Y 140.531,Z 382.251,A -85,B 0,C 180,E1 -27188.624,E2 -27188.624} C_VEL
LIN {X 0,Y 139.799,Z 382.129,A -85,B 0,C 180,E1 -27197.55,E2 -27197.55} C_VEL
LIN {X 0,Y 140.209,Z 382.479,A -85,B 0,C 180,E1 -27200.732,E2 -27200.732} C_VEL
LIN {X 0,Y 141.324,Z 385.507,A -85,B 0,C 180,E1 -27205.842,E2 -27205.842} C_VEL
LIN {X 0,Y 142.658,Z 387.209,A -85,B 0,C 180,E1 -27209.173,E2 -27209.173} C_VEL
LIN {X 0,Y 145.205,Z 391.555,A -85,B 0,C 180,E1 -27214.142,E2 -27214.142} C_VEL
LIN {X 0,Y 147.705,Z 395.884,A -85,B 0,C 180,E1 -27217.858,E2 -27217.858} C_VEL
LIN {X 0,Y 150.76,Z 401.214,A -85,B 0,C 180,E1 -27221.66,E2 -27221.66} C_VEL
LIN {X 0,Y 154.485,Z 408.319,A -85,B 0,C 180,E1 -27225.572,E2 -27225.572} C_VEL
LIN {X 0,Y 158.636,Z 416.921,A -85,B 0,C 180,E1 -27229.349,E2 -27229.349} C_VEL
LIN {X 0,Y 161.226,Z 422.639,A -85,B 0,C 180,E1 -27231.472,E2 -27231.472} C_VEL
LIN {X 0,Y 155.777,Z 471.524,A -85,B 0,C 180,E1 -27233.075,E2 -27233.075} C_VEL
LIN {X 0,Y 152.764,Z 487.346,A -85,B 0,C 180,E1 -27233.882,E2 -27233.882} C_VEL
LIN {X 0,Y 148.733,Z 502.593,A -85,B 0,C 180,E1 -27235.044,E2 -27235.044} C_VEL
LIN {X 0,Y 144.338,Z 515.554,A -85,B 0,C 180,E1 -27236.35,E2 -27236.35} C_VEL
LIN {X 0,Y 138.596,Z 529.564,A -85,B 0,C 180,E1 -27238.257,E2 -27238.257} C_VEL
LIN {X 0,Y 131.569,Z 543.739,A -85,B 0,C 180,E1 -27240.828,E2 -27240.828} C_VEL
LIN {X 0,Y 124.78,Z 555.527,A -85,B 0,C 180,E1 -27243.669,E2 -27243.669} C_VEL
LIN {X 0,Y 117.668,Z 566.45,A -85,B 0,C 180,E1 -27247.155,E2 -27247.155} C_VEL
LIN {X 0,Y 110.491,Z 576.48,A -85,B 0,C 180,E1 -27251.455,E2 -27251.455} C_VEL
LIN {X 0,Y 102.852,Z 586.3,A -85,B 0,C 180,E1 -27257.168,E2 -27257.168} C_VEL
LIN {X 0,Y 96.236,Z 594.393,A -85,B 0,C 180,E1 -27263.709,E2 -27263.709} C_VEL
LIN {X 0,Y 91.352,Z 600.389,A -85,B 0,C 180,E1 -27270.32,E2 -27270.32} C_VEL
LIN {X 0,Y 86.929,Z 606.335,A -85,B 0,C 180,E1 -27279.303,E2 -27279.303} C_VEL
LIN {X 0,Y 84.626,Z 610,A -85,B 0,C 180,E1 -27286.896,E2 -27286.896} C_VEL
LIN {X 0,Y 83.256,Z 612.826,A -85,B 0,C 180,E1 -27294.963,E2 -27294.963} C_VEL
LIN {X 0,Y 83.146,Z 614.675,A -85,B 0,C 180,E1 -27302.317,E2 -27302.317} C_VEL
LIN {X 0,Y 84.4,Z 616.047,A -85,B 0,C 180,E1 -27311.768,E2 -27311.768} C_VEL
LIN {X 0,Y 86.882,Z 616.377,A -85,B 0,C 180,E1 -27319.685,E2 -27319.685} C_VEL
LIN {X 0,Y 91.178,Z 615.849,A -85,B 0,C 180,E1 -27327.977,E2 -27327.977} C_VEL
LIN {X 0,Y 95.607,Z 614.709,A -85,B 0,C 180,E1 -27333.837,E2 -27333.837} C_VEL
LIN {X 0,Y 103.682,Z 611.934,A -85,B 0,C 180,E1 -27341.609,E2 -27341.609} C_VEL
LIN {X 0,Y 111.706,Z 608.518,A -85,B 0,C 180,E1 -27347.196,E2 -27347.196} C_VEL
LIN {X 0,Y 120.651,Z 604.02,A -85,B 0,C 180,E1 -27351.977,E2 -27351.977} C_VEL
LIN {X 0,Y 129.956,Z 598.673,A -85,B 0,C 180,E1 -27355.9,E2 -27355.9} C_VEL
LIN {X 0,Y 140.559,Z 591.612,A -85,B 0,C 180,E1 -27359.517,E2 -27359.517} C_VEL
LIN {X 0,Y 151.856,Z 582.802,A -85,B 0,C 180,E1 -27362.657,E2 -27362.657} C_VEL
LIN {X 0,Y 162.275,Z 573.397,A -85,B 0,C 180,E1 -27365.08,E2 -27365.08} C_VEL
LIN {X 0,Y 172.147,Z 563.032,A -85,B 0,C 180,E1 -27367.039,E2 -27367.039} C_VEL
LIN {X 0,Y 181.679,Z 551.295,A -85,B 0,C 180,E1 -27368.702,E2 -27368.702} C_VEL
LIN {X 0,Y 189.993,Z 539.205,A -85,B 0,C 180,E1 -27369.988,E2 -27369.988} C_VEL
LIN {X 0,Y 198.089,Z 525.187,A -85,B 0,C 180,E1 -27371.134,E2 -27371.134} C_VEL
LIN {X 0,Y 204.803,Z 510.804,A -85,B 0,C 180,E1 -27372.006,E2 -27372.006} C_VEL
LIN {X 0,Y 210.39,Z 495.437,A -85,B 0,C 180,E1 -27372.692,E2 -27372.692} C_VEL
LIN {X 0,Y 214.367,Z 480.729,A -85,B 0,C 180,E1 -27373.15,E2 -27373.15} C_VEL
LIN {X 0,Y 217.277,Z 464.44,A -85,B 0,C 180,E1 -27373.511,E2 -27373.511} C_VEL
LIN {X 0,Y 217.685,Z 461.415,A -85,B 0,C 180,E1 -27373.637,E2 -27373.637} C_VEL
LIN {X 0,Y 217.683,Z 461.533,A -85,B 0,C 180,E1 -27376.084,E2 -27376.084} C_VEL
LIN {X 0,Y 214.715,Z 479.215,A -85,B 0,C 180,E1 -27376.475,E2 -27376.475} C_VEL
LIN {X 0,Y 210.588,Z 495.035,A -85,B 0,C 180,E1 -27376.888,E2 -27376.888} C_VEL
LIN {X 0,Y 205.319,Z 509.844,A -85,B 0,C 180,E1 -27377.424,E2 -27377.424} C_VEL
LIN {X 0,Y 198.744,Z 524.32,A -85,B 0,C 180,E1 -27378.136,E2 -27378.136} C_VEL
LIN {X 0,Y 192.195,Z 536.132,A -85,B 0,C 180,E1 -27378.891,E2 -27378.891} C_VEL
LIN {X 0,Y 183.347,Z 549.653,A -85,B 0,C 180,E1 -27380.104,E2 -27380.104} C_VEL
LIN {X 0,Y 173.802,Z 561.907,A -85,B 0,C 180,E1 -27381.564,E2 -27381.564} C_VEL
LIN {X 0,Y 164.458,Z 572.216,A -85,B 0,C 180,E1 -27383.256,E2 -27383.256} C_VEL
LIN {X 0,Y 156.811,Z 579.67,A -85,B 0,C 180,E1 -27384.833,E2 -27384.833} C_VEL
LIN {X 0,Y 146.322,Z 588.659,A -85,B 0,C 180,E1 -27387.31,E2 -27387.31} C_VEL
LIN {X 0,Y 134.84,Z 597.22,A -85,B 0,C 180,E1 -27390.688,E2 -27390.688} C_VEL
LIN {X 0,Y 124.023,Z 604.155,A -85,B 0,C 180,E1 -27394.684,E2 -27394.684} C_VEL
LIN {X 0,Y 113.96,Z 609.79,A -85,B 0,C 180,E1 -27399.57,E2 -27399.57} C_VEL
LIN {X 0,Y 107.017,Z 613.199,A -85,B 0,C 180,E1 -27403.751,E2 -27403.751} C_VEL
LIN {X 0,Y 98.849,Z 616.678,A -85,B 0,C 180,E1 -27410.22,E2 -27410.22} C_VEL
LIN {X 0,Y 92.219,Z 619.06,A -85,B 0,C 180,E1 -27417.763,E2 -27417.763} C_VEL
LIN {X 0,Y 87.404,Z 620.391,A -85,B 0,C 180,E1 -27426.297,E2 -27426.297} C_VEL
LIN {X 0,Y 84.597,Z 620.593,A -85,B 0,C 180,E1 -27435.57,E2 -27435.57} C_VEL
LIN {X 0,Y 83.76,Z 619.728,A -85,B 0,C 180,E1 -27445.189,E2 -27445.189} C_VEL
LIN {X 0,Y 83.907,Z 618.877,A -85,B 0,C 180,E1 -27450.002,E2 -27450.002} C_VEL
LIN {X 0,Y 83.994,Z 616.183,A -85,B 0,C 180,E1 -27459.635,E2 -27459.635} C_VEL
LIN {X 0,Y 85.679,Z 612.165,A -85,B 0,C 180,E1 -27469.155,E2 -27469.155} C_VEL
LIN {X 0,Y 87.035,Z 609.959,A -85,B 0,C 180,E1 -27473.16,E2 -27473.16} C_VEL
LIN {X 0,Y 87.871,Z 607.827,A -85,B 0,C 180,E1 -27476.728,E2 -27476.728} C_VEL
LIN {X 0,Y 88.142,Z 603.829,A -85,B 0,C 180,E1 -27482.639,E2 -27482.639} C_VEL
LIN {X 0,Y 89.171,Z 599.37,A -85,B 0,C 180,E1 -27488.336,E2 -27488.336} C_VEL
LIN {X 0,Y 91.115,Z 596.389,A -85,B 0,C 180,E1 -27491.369,E2 -27491.369} C_VEL
LIN {X 0,Y 99.012,Z 587.266,A -85,B 0,C 180,E1 -27498.186,E2 -27498.186} C_VEL
LIN {X 0,Y 107.081,Z 577.009,A -85,B 0,C 180,E1 -27503.632,E2 -27503.632} C_VEL
LIN {X 0,Y 114.608,Z 566.759,A -85,B 0,C 180,E1 -27507.478,E2 -27507.478} C_VEL
LIN {X 0,Y 122.663,Z 554.401,A -85,B 0,C 180,E1 -27510.898,E2 -27510.898} C_VEL
LIN {X 0,Y 128.967,Z 543.308,A -85,B 0,C 180,E1 -27513.17,E2 -27513.17} C_VEL
LIN {X 0,Y 135.074,Z 530.956,A -85,B 0,C 180,E1 -27515.108,E2 -27515.108} C_VEL
LIN {X 0,Y 140.999,Z 516.669,A -85,B 0,C 180,E1 -27516.781,E2 -27516.781} C_VEL
LIN {X 0,Y 145.911,Z 502.043,A -85,B 0,C 180,E1 -27518.003,E2 -27518.003} C_VEL
LIN {X 0,Y 149.709,Z 487.036,A -85,B 0,C 180,E1 -27518.91,E2 -27518.91} C_VEL
LIN {X 0,Y 152.37,Z 471.508,A -85,B 0,C 180,E1 -27519.564,E2 -27519.564} C_VEL
LIN {X 0,Y 157.274,Z 428.362,A -85,B 0,C 180,E1 -27520.891,E2 -27520.891} C_VEL
LIN {X 0,Y 154.05,Z 418.46,A -85,B 0,C 180,E1 -27524.11,E2 -27524.11} C_VEL
LIN {X 0,Y 149.942,Z 409.905,A -85,B 0,C 180,E1 -27528.436,E2 -27528.436} C_VEL
LIN {X 0,Y 146.246,Z 402.658,A -85,B 0,C 180,E1 -27533.187,E2 -27533.187} C_VEL
LIN {X 0,Y 144.475,Z 399.441,A -85,B 0,C 180,E1 -27535.848,E2 -27535.848} C_VEL
LIN {X 0,Y 142.722,Z 396.022,A -85,B 0,C 180,E1 -27539.079,E2 -27539.079} C_VEL
LIN {X 0,Y 141.104,Z 392.777,A -85,B 0,C 180,E1 -27542.85,E2 -27542.85} C_VEL
LIN {X 0,Y 139.509,Z 389.401,A -85,B 0,C 180,E1 -27548.687,E2 -27548.687} C_VEL
LIN {X 0,Y 138.761,Z 389.078,A -85,B 0,C 180,E1 -27555.78,E2 -27555.78} C_VEL
LIN {X 0,Y 139.147,Z 389.552,A -85,B 0,C 180,E1 -27560.387,E2 -27560.387} C_VEL
LIN {X 0,Y 140.5,Z 392.886,A -85,B 0,C 180,E1 -27566.38,E2 -27566.38} C_VEL
LIN {X 0,Y 141.315,Z 393.99,A -85,B 0,C 180,E1 -27568.467,E2 -27568.467} C_VEL
LIN {X 0,Y 143.68,Z 398.275,A -85,B 0,C 180,E1 -27573.388,E2 -27573.388} C_VEL
LIN {X 0,Y 145.958,Z 402.4,A -85,B 0,C 180,E1 -27576.988,E2 -27576.988} C_VEL
LIN {X 0,Y 148.851,Z 407.812,A -85,B 0,C 180,E1 -27580.823,E2 -27580.823} C_VEL
LIN {X 0,Y 152.587,Z 415.222,A -85,B 0,C 180,E1 -27584.931,E2 -27584.931} C_VEL
LIN {X 0,Y 156.855,Z 424.807,A -85,B 0,C 180,E1 -27589.017,E2 -27589.017} C_VEL
LIN {X 0,Y 157.306,Z 425.883,A -85,B 0,C 180,E1 -27589.414,E2 -27589.414} C_VEL
LIN {X 0,Y 151.991,Z 471.601,A -85,B 0,C 180,E1 -27590.843,E2 -27590.843} C_VEL
LIN {X 0,Y 148.902,Z 487.454,A -85,B 0,C 180,E1 -27591.63,E2 -27591.63} C_VEL
LIN {X 0,Y 144.953,Z 502.068,A -85,B 0,C 180,E1 -27592.695,E2 -27592.695} C_VEL
LIN {X 0,Y 140.062,Z 516.095,A -85,B 0,C 180,E1 -27594.073,E2 -27594.073} C_VEL
LIN {X 0,Y 134.504,Z 529.237,A -85,B 0,C 180,E1 -27595.826,E2 -27595.826} C_VEL
LIN {X 0,Y 127.926,Z 542.227,A -85,B 0,C 180,E1 -27598.076,E2 -27598.076} C_VEL
LIN {X 0,Y 119.959,Z 555.691,A -85,B 0,C 180,E1 -27601.235,E2 -27601.235} C_VEL
LIN {X 0,Y 112.086,Z 567.257,A -85,B 0,C 180,E1 -27604.96,E2 -27604.96} C_VEL
LIN {X 0,Y 104.74,Z 577.007,A -85,B 0,C 180,E1 -27609.242,E2 -27609.242} C_VEL
LIN {X 0,Y 96.552,Z 586.928,A -85,B 0,C 180,E1 -27615.239,E2 -27615.239} C_VEL
LIN {X 0,Y 89.578,Z 594.95,A -85,B 0,C 180,E1 -27622.107,E2 -27622.107} C_VEL
LIN {X 0,Y 83.92,Z 601.504,A -85,B 0,C 180,E1 -27629.998,E2 -27629.998} C_VEL
LIN {X 0,Y 80.291,Z 606.076,A -85,B 0,C 180,E1 -27637.542,E2 -27637.542} C_VEL
LIN {X 0,Y 77.716,Z 609.86,A -85,B 0,C 180,E1 -27645.739,E2 -27645.739} C_VEL
LIN {X 0,Y 76.338,Z 612.328,A -85,B 0,C 180,E1 -27653.004,E2 -27653.004} C_VEL
LIN {X 0,Y 76.105,Z 614.927,A -85,B 0,C 180,E1 -27663.804,E2 -27663.804} C_VEL
LIN {X 0,Y 77.623,Z 616.238,A -85,B 0,C 180,E1 -27673.601,E2 -27673.601} C_VEL
LIN {X 0,Y 80.644,Z 616.595,A -85,B 0,C 180,E1 -27682.419,E2 -27682.419} C_VEL
LIN {X 0,Y 86.856,Z 615.792,A -85,B 0,C 180,E1 -27692.876,E2 -27692.876} C_VEL
LIN {X 0,Y 91.097,Z 614.776,A -85,B 0,C 180,E1 -27697.779,E2 -27697.779} C_VEL
LIN {X 0,Y 96.944,Z 613.003,A -85,B 0,C 180,E1 -27703.151,E2 -27703.151} C_VEL
LIN {X 0,Y 107.041,Z 609.175,A -85,B 0,C 180,E1 -27709.999,E2 -27709.999} C_VEL
LIN {X 0,Y 116.453,Z 604.852,A -85,B 0,C 180,E1 -27714.709,E2 -27714.709} C_VEL
LIN {X 0,Y 126.533,Z 599.444,A -85,B 0,C 180,E1 -27718.668,E2 -27718.668} C_VEL
LIN {X 0,Y 138.511,Z 591.834,A -85,B 0,C 180,E1 -27722.419,E2 -27722.419} C_VEL
LIN {X 0,Y 150.206,Z 583.072,A -85,B 0,C 180,E1 -27725.374,E2 -27725.374} C_VEL
LIN {X 0,Y 161.487,Z 573.13,A -85,B 0,C 180,E1 -27727.717,E2 -27727.717} C_VEL
LIN {X 0,Y 171.223,Z 563.123,A -85,B 0,C 180,E1 -27729.454,E2 -27729.454} C_VEL
LIN {X 0,Y 180.953,Z 551.451,A -85,B 0,C 180,E1 -27730.981,E2 -27730.981} C_VEL
LIN {X 0,Y 190.281,Z 538.105,A -85,B 0,C 180,E1 -27732.26,E2 -27732.26} C_VEL
LIN {X 0,Y 197.604,Z 525.525,A -85,B 0,C 180,E1 -27733.198,E2 -27733.198} C_VEL
LIN {X 0,Y 204.586,Z 510.782,A -85,B 0,C 180,E1 -27734.011,E2 -27734.011} C_VEL
LIN {X 0,Y 210.149,Z 495.675,A -85,B 0,C 180,E1 -27734.633,E2 -27734.633} C_VEL
LIN {X 0,Y 211.789,Z 490.233,A -85,B 0,C 180,E1 -27734.794,E2 -27734.794} C_VEL
LIN {X 0,Y 206.663,Z 505.63,A -85,B 0,C 180,E1 -27735.276,E2 -27735.276} C_VEL
LIN {X 0,Y 200.874,Z 519.178,A -85,B 0,C 180,E1 -27735.823,E2 -27735.823} C_VEL
LIN {X 0,Y 193.38,Z 533.287,A -85,B 0,C 180,E1 -27736.562,E2 -27736.562} C_VEL
LIN {X 0,Y 184.347,Z 547.217,A -85,B 0,C 180,E1 -27737.625,E2 -27737.625} C_VEL
LIN {X 0,Y 174.728,Z 559.628,A -85,B 0,C 180,E1 -27738.922,E2 -27738.922} C_VEL
LIN {X 0,Y 164.974,Z 570.4,A -85,B 0,C 180,E1 -27740.417,E2 -27740.417} C_VEL
LIN {X 0,Y 154,Z 580.822,A -85,B 0,C 180,E1 -27742.467,E2 -27742.467} C_VEL
LIN {X 0,Y 143.231,Z 589.592,A -85,B 0,C 180,E1 -27744.809,E2 -27744.809} C_VEL
LIN {X 0,Y 131.378,Z 597.905,A -85,B 0,C 180,E1 -27748.04,E2 -27748.04} C_VEL
LIN {X 0,Y 119.717,Z 604.903,A -85,B 0,C 180,E1 -27752.06,E2 -27752.06} C_VEL
LIN {X 0,Y 109.567,Z 610.128,A -85,B 0,C 180,E1 -27756.702,E2 -27756.702} C_VEL
LIN {X 0,Y 102.199,Z 613.441,A -85,B 0,C 180,E1 -27760.852,E2 -27760.852} C_VEL
LIN {X 0,Y 93.478,Z 616.774,A -85,B 0,C 180,E1 -27767.421,E2 -27767.421} C_VEL
LIN {X 0,Y 86.232,Z 619.02,A -85,B 0,C 180,E1 -27775.217,E2 -27775.217} C_VEL
LIN {X 0,Y 80.892,Z 620.223,A -85,B 0,C 180,E1 -27784.255,E2 -27784.255} C_VEL
LIN {X 0,Y 77.68,Z 620.357,A -85,B 0,C 180,E1 -27794.254,E2 -27794.254} C_VEL
LIN {X 0,Y 76.675,Z 619.37,A -85,B 0,C 180,E1 -27804.743,E2 -27804.743} C_VEL
LIN {X 0,Y 76.803,Z 618.456,A -85,B 0,C 180,E1 -27810.002,E2 -27810.002} C_VEL
LIN {X 0,Y 76.692,Z 617.206,A -85,B 0,C 180,E1 -27815.26,E2 -27815.26} C_VEL
LIN {X 0,Y 77.728,Z 613.734,A -85,B 0,C 180,E1 -27825.741,E2 -27825.741} C_VEL
LIN {X 0,Y 80.744,Z 608.884,A -85,B 0,C 180,E1 -27835.8,E2 -27835.8} C_VEL
LIN {X 0,Y 86.001,Z 602.346,A -85,B 0,C 180,E1 -27845.183,E2 -27845.183} C_VEL
LIN {X 0,Y 91.115,Z 596.389,A -85,B 0,C 180,E1 -27851.369,E2 -27851.369} C_VEL
LIN {X 0,Y 93.234,Z 593.306,A -85,B 0,C 180,E1 -27854.216,E2 -27854.216} C_VEL
LIN {X 0,Y 95.52,Z 587.86,A -85,B 0,C 180,E1 -27859.061,E2 -27859.061} C_VEL
LIN {X 0,Y 98.21,Z 582.038,A -85,B 0,C 180,E1 -27863.532,E2 -27863.532} C_VEL
LIN {X 0,Y 100.837,Z 578.193,A -85,B 0,C 180,E1 -27865.684,E2 -27865.684} C_VEL
LIN {X 0,Y 108.184,Z 568.796,A -85,B 0,C 180,E1 -27869.403,E2 -27869.403} C_VEL
LIN {X 0,Y 116.48,Z 556.88,A -85,B 0,C 180,E1 -27872.869,E2 -27872.869} C_VEL
LIN {X 0,Y 123.69,Z 545.027,A -85,B 0,C 180,E1 -27875.383,E2 -27875.383} C_VEL
LIN {X 0,Y 130.699,Z 531.528,A -85,B 0,C 180,E1 -27877.503,E2 -27877.503} C_VEL
LIN {X 0,Y 136.411,Z 518.376,A -85,B 0,C 180,E1 -27879.038,E2 -27879.038} C_VEL
LIN {X 0,Y 141.433,Z 504.297,A -85,B 0,C 180,E1 -27880.226,E2 -27880.226} C_VEL
LIN {X 0,Y 145.511,Z 489.333,A -85,B 0,C 180,E1 -27881.148,E2 -27881.148} C_VEL
LIN {X 0,Y 148.388,Z 474.418,A -85,B 0,C 180,E1 -27881.778,E2 -27881.778} C_VEL
LIN {X 0,Y 153.491,Z 430.969,A -85,B 0,C 180,E1 -27883.111,E2 -27883.111} C_VEL
LIN {X 0,Y 151.316,Z 423.811,A -85,B 0,C 180,E1 -27885.554,E2 -27885.554} C_VEL
LIN {X 0,Y 147.72,Z 415.856,A -85,B 0,C 180,E1 -27889.632,E2 -27889.632} C_VEL
LIN {X 0,Y 143.971,Z 408.103,A -85,B 0,C 180,E1 -27894.893,E2 -27894.893} C_VEL
LIN {X 0,Y 141.3,Z 402.682,A -85,B 0,C 180,E1 -27899.863,E2 -27899.863} C_VEL
LIN {X 0,Y 139.805,Z 399.538,A -85,B 0,C 180,E1 -27903.583,E2 -27903.583} C_VEL
LIN {X 0,Y 138.356,Z 396.274,A -85,B 0,C 180,E1 -27909.458,E2 -27909.458} C_VEL
LIN {X 0,Y 137.855,Z 396.191,A -85,B 0,C 180,E1 -27917.806,E2 -27917.806} C_VEL
LIN {X 0,Y 138.086,Z 396.513,A -85,B 0,C 180,E1 -27919.923,E2 -27919.923} C_VEL
LIN {X 0,Y 139.279,Z 399.723,A -85,B 0,C 180,E1 -27925.749,E2 -27925.749} C_VEL
LIN {X 0,Y 140.057,Z 400.94,A -85,B 0,C 180,E1 -27927.929,E2 -27927.929} C_VEL
LIN {X 0,Y 142.171,Z 404.926,A -85,B 0,C 180,E1 -27932.588,E2 -27932.588} C_VEL
LIN {X 0,Y 144.917,Z 410.176,A -85,B 0,C 180,E1 -27937.107,E2 -27937.107} C_VEL
LIN {X 0,Y 148.062,Z 416.59,A -85,B 0,C 180,E1 -27941.316,E2 -27941.316} C_VEL
LIN {X 0,Y 151.608,Z 424.411,A -85,B 0,C 180,E1 -27945.272,E2 -27945.272} C_VEL
LIN {X 0,Y 153.511,Z 429.324,A -85,B 0,C 180,E1 -27947.246,E2 -27947.246} C_VEL
LIN {X 0,Y 148.256,Z 472.473,A -85,B 0,C 180,E1 -27948.533,E2 -27948.533} C_VEL
LIN {X 0,Y 145.13,Z 487.974,A -85,B 0,C 180,E1 -27949.29,E2 -27949.29} C_VEL
LIN {X 0,Y 141.046,Z 502.591,A -85,B 0,C 180,E1 -27950.326,E2 -27950.326} C_VEL
LIN {X 0,Y 135.977,Z 516.644,A -85,B 0,C 180,E1 -27951.667,E2 -27951.667} C_VEL
LIN {X 0,Y 129.904,Z 530.453,A -85,B 0,C 180,E1 -27953.478,E2 -27953.478} C_VEL
LIN {X 0,Y 123.111,Z 543.288,A -85,B 0,C 180,E1 -27955.685,E2 -27955.685} C_VEL
LIN {X 0,Y 115.152,Z 556.131,A -85,B 0,C 180,E1 -27958.686,E2 -27958.686} C_VEL
LIN {X 0,Y 106.67,Z 568.016,A -85,B 0,C 180,E1 -27962.535,E2 -27962.535} C_VEL
LIN {X 0,Y 98.238,Z 578.583,A -85,B 0,C 180,E1 -27967.356,E2 -27967.356} C_VEL
LIN {X 0,Y 90.373,Z 587.523,A -85,B 0,C 180,E1 -27973.043,E2 -27973.043} C_VEL
LIN {X 0,Y 83.019,Z 595.477,A -85,B 0,C 180,E1 -27980.25,E2 -27980.25} C_VEL
LIN {X 0,Y 77.336,Z 601.608,A -85,B 0,C 180,E1 -27988.124,E2 -27988.124} C_VEL
LIN {X 0,Y 72.656,Z 607.194,A -85,B 0,C 180,E1 -27998.34,E2 -27998.34} C_VEL
LIN {X 0,Y 70.123,Z 610.758,A -85,B 0,C 180,E1 -28007.495,E2 -28007.495} C_VEL
LIN {X 0,Y 69.12,Z 612.687,A -85,B 0,C 180,E1 -28013.996,E2 -28013.996} C_VEL
LIN {X 0,Y 69.127,Z 615.171,A -85,B 0,C 180,E1 -28025.594,E2 -28025.594} C_VEL
LIN {X 0,Y 71.077,Z 616.462,A -85,B 0,C 180,E1 -28036.213,E2 -28036.213} C_VEL
LIN {X 0,Y 75.351,Z 616.788,A -85,B 0,C 180,E1 -28047.074,E2 -28047.074} C_VEL
LIN {X 0,Y 79.583,Z 616.378,A -85,B 0,C 180,E1 -28053.807,E2 -28053.807} C_VEL
LIN {X 0,Y 88.144,Z 614.589,A -85,B 0,C 180,E1 -28063.086,E2 -28063.086} C_VEL
LIN {X 0,Y 93.603,Z 613.033,A -85,B 0,C 180,E1 -28067.428,E2 -28067.428} C_VEL
LIN {X 0,Y 100.769,Z 610.587,A -85,B 0,C 180,E1 -28071.989,E2 -28071.989} C_VEL
LIN {X 0,Y 112.537,Z 605.68,A -85,B 0,C 180,E1 -28077.654,E2 -28077.654} C_VEL
LIN {X 0,Y 124.82,Z 599.438,A -85,B 0,C 180,E1 -28082.034,E2 -28082.034} C_VEL
LIN {X 0,Y 136.26,Z 592.502,A -85,B 0,C 180,E1 -28085.249,E2 -28085.249} C_VEL
LIN {X 0,Y 149.094,Z 583.191,A -85,B 0,C 180,E1 -28088.166,E2 -28088.166} C_VEL
LIN {X 0,Y 159.691,Z 574.211,A -85,B 0,C 180,E1 -28090.143,E2 -28090.143} C_VEL
LIN {X 0,Y 170.68,Z 563.267,A -85,B 0,C 180,E1 -28091.885,E2 -28091.885} C_VEL
LIN {X 0,Y 180.503,Z 551.7,A -85,B 0,C 180,E1 -28093.256,E2 -28093.256} C_VEL
LIN {X 0,Y 188.531,Z 540.539,A -85,B 0,C 180,E1 -28094.261,E2 -28094.261} C_VEL
LIN {X 0,Y 189.697,Z 538.817,A -85,B 0,C 180,E1 -28094.383,E2 -28094.383} C_VEL
LIN {X 0,Y 189.042,Z 539.827,A -85,B 0,C 180,E1 -28094.858,E2 -28094.858} C_VEL
LIN {X 0,Y 180.719,Z 551.568,A -85,B 0,C 180,E1 -28095.763,E2 -28095.763} C_VEL
LIN {X 0,Y 170.967,Z 563.231,A -85,B 0,C 180,E1 -28096.963,E2 -28096.963} C_VEL
LIN {X 0,Y 161.07,Z 573.345,A -85,B 0,C 180,E1 -28098.38,E2 -28098.38} C_VEL
LIN {X 0,Y 151.463,Z 581.894,A -85,B 0,C 180,E1 -28100.019,E2 -28100.019} C_VEL
LIN {X 0,Y 140.426,Z 590.471,A -85,B 0,C 180,E1 -28102.204,E2 -28102.204} C_VEL
LIN {X 0,Y 128.213,Z 598.589,A -85,B 0,C 180,E1 -28105.257,E2 -28105.257} C_VEL
LIN {X 0,Y 115.673,Z 605.599,A -85,B 0,C 180,E1 -28109.25,E2 -28109.25} C_VEL
LIN {X 0,Y 105.472,Z 610.477,A -85,B 0,C 180,E1 -28113.605,E2 -28113.605} C_VEL
LIN {X 0,Y 97.67,Z 613.646,A -85,B 0,C 180,E1 -28117.676,E2 -28117.676} C_VEL
LIN {X 0,Y 88.349,Z 616.883,A -85,B 0,C 180,E1 -28124.284,E2 -28124.284} C_VEL
LIN {X 0,Y 80.448,Z 618.981,A -85,B 0,C 180,E1 -28132.304,E2 -28132.304} C_VEL
LIN {X 0,Y 74.507,Z 620.049,A -85,B 0,C 180,E1 -28141.863,E2 -28141.863} C_VEL
LIN {X 0,Y 70.817,Z 620.091,A -85,B 0,C 180,E1 -28152.682,E2 -28152.682} C_VEL
LIN {X 0,Y 69.583,Z 619.01,A -85,B 0,C 180,E1 -28164.206,E2 -28164.206} C_VEL
LIN {X 0,Y 69.716,Z 618.037,A -85,B 0,C 180,E1 -28170.002,E2 -28170.002} C_VEL
LIN {X 0,Y 69.964,Z 615.084,A -85,B 0,C 180,E1 -28181.592,E2 -28181.592} C_VEL
LIN {X 0,Y 72.295,Z 610.797,A -85,B 0,C 180,E1 -28192.885,E2 -28192.885} C_VEL
LIN {X 0,Y 76.933,Z 605.068,A -85,B 0,C 180,E1 -28203.239,E2 -28203.239} C_VEL
LIN {X 0,Y 83.626,Z 597.744,A -85,B 0,C 180,E1 -28212.248,E2 -28212.248} C_VEL
LIN {X 0,Y 90.924,Z 589.875,A -85,B 0,C 180,E1 -28218.907,E2 -28218.907} C_VEL
LIN {X 0,Y 99.117,Z 580.335,A -85,B 0,C 180,E1 -28224.63,E2 -28224.63} C_VEL
LIN {X 0,Y 100.837,Z 578.193,A -85,B 0,C 180,E1 -28225.684,E2 -28225.684} C_VEL
LIN {X 0,Y 103.52,Z 574.288,A -85,B 0,C 180,E1 -28227.664,E2 -28227.664} C_VEL
LIN {X 0,Y 106.756,Z 567.578,A -85,B 0,C 180,E1 -28231.229,E2 -28231.229} C_VEL
LIN {X 0,Y 110.065,Z 560.51,A -85,B 0,C 180,E1 -28234.466,E2 -28234.466} C_VEL
LIN {X 0,Y 112.712,Z 555.979,A -85,B 0,C 180,E1 -28235.884,E2 -28235.884} C_VEL
LIN {X 0,Y 120.104,Z 544.115,A -85,B 0,C 180,E1 -28238.27,E2 -28238.27} C_VEL
LIN {X 0,Y 126.993,Z 531.187,A -85,B 0,C 180,E1 -28240.188,E2 -28240.188} C_VEL
LIN {X 0,Y 133.219,Z 517.101,A -85,B 0,C 180,E1 -28241.731,E2 -28241.731} C_VEL
LIN {X 0,Y 138.371,Z 502.714,A -85,B 0,C 180,E1 -28242.843,E2 -28242.843} C_VEL
LIN {X 0,Y 142.352,Z 488.114,A -85,B 0,C 180,E1 -28243.666,E2 -28243.666} C_VEL
LIN {X 0,Y 145.129,Z 473.61,A -85,B 0,C 180,E1 -28244.251,E2 -28244.251} C_VEL
LIN {X 0,Y 149.963,Z 433.561,A -85,B 0,C 180,E1 -28245.436,E2 -28245.436} C_VEL
LIN {X 0,Y 148.428,Z 428.594,A -85,B 0,C 180,E1 -28247.297,E2 -28247.297} C_VEL
LIN {X 0,Y 145.358,Z 421.456,A -85,B 0,C 180,E1 -28251.13,E2 -28251.13} C_VEL
LIN {X 0,Y 142.12,Z 414.269,A -85,B 0,C 180,E1 -28256.099,E2 -28256.099} C_VEL
LIN {X 0,Y 139.825,Z 409.256,A -85,B 0,C 180,E1 -28260.805,E2 -28260.805} C_VEL
LIN {X 0,Y 138.543,Z 406.325,A -85,B 0,C 180,E1 -28264.285,E2 -28264.285} C_VEL
LIN {X 0,Y 137.346,Z 403.36,A -85,B 0,C 180,E1 -28269.528,E2 -28269.528} C_VEL
LIN {X 0,Y 136.883,Z 403.231,A -85,B 0,C 180,E1 -28277.937,E2 -28277.937} C_VEL
LIN {X 0,Y 137.043,Z 403.545,A -85,B 0,C 180,E1 -28279.569,E2 -28279.569} C_VEL
LIN {X 0,Y 138.379,Z 406.992,A -85,B 0,C 180,E1 -28286.072,E2 -28286.072} C_VEL
LIN {X 0,Y 138.976,Z 408.249,A -85,B 0,C 180,E1 -28287.842,E2 -28287.842} C_VEL
LIN {X 0,Y 140.619,Z 411.456,A -85,B 0,C 180,E1 -28291.631,E2 -28291.631} C_VEL
LIN {X 0,Y 142.827,Z 416.047,A -85,B 0,C 180,E1 -28295.669,E2 -28295.669} C_VEL
LIN {X 0,Y 145.276,Z 421.278,A -85,B 0,C 180,E1 -28299.283,E2 -28299.283} C_VEL
LIN {X 0,Y 148.393,Z 428.542,A -85,B 0,C 180,E1 -28303.202,E2 -28303.202} C_VEL
LIN {X 0,Y 149.923,Z 432.243,A -85,B 0,C 180,E1 -28304.894,E2 -28304.894} C_VEL
LIN {X 0,Y 144.945,Z 472.474,A -85,B 0,C 180,E1 -28306.086,E2 -28306.086} C_VEL
LIN {X 0,Y 141.786,Z 487.839,A -85,B 0,C 180,E1 -28306.791,E2 -28306.791} C_VEL
LIN {X 0,Y 137.402,Z 503.103,A -85,B 0,C 180,E1 -28307.829,E2 -28307.829} C_VEL
LIN {X 0,Y 132.584,Z 516.149,A -85,B 0,C 180,E1 -28309.006,E2 -28309.006} C_VEL
LIN {X 0,Y 126.495,Z 529.727,A -85,B 0,C 180,E1 -28310.692,E2 -28310.692} C_VEL
LIN {X 0,Y 119.313,Z 542.986,A -85,B 0,C 180,E1 -28312.859,E2 -28312.859} C_VEL
LIN {X 0,Y 111.7,Z 554.951,A -85,B 0,C 180,E1 -28315.509,E2 -28315.509} C_VEL
LIN {X 0,Y 104.335,Z 565.088,A -85,B 0,C 180,E1 -28318.53,E2 -28318.53} C_VEL
LIN {X 0,Y 95.956,Z 575.433,A -85,B 0,C 180,E1 -28322.756,E2 -28322.756} C_VEL
LIN {X 0,Y 88.079,Z 584.199,A -85,B 0,C 180,E1 -28327.726,E2 -28327.726} C_VEL
LIN {X 0,Y 79.729,Z 592.769,A -85,B 0,C 180,E1 -28334.664,E2 -28334.664} C_VEL
LIN {X 0,Y 73.589,Z 598.925,A -85,B 0,C 180,E1 -28341.762,E2 -28341.762} C_VEL
LIN {X 0,Y 68.63,Z 604.003,A -85,B 0,C 180,E1 -28349.998,E2 -28349.998} C_VEL
LIN {X 0,Y 64.435,Z 608.869,A -85,B 0,C 180,E1 -28361.054,E2 -28361.054} C_VEL
LIN {X 0,Y 62.505,Z 611.632,A -85,B 0,C 180,E1 -28369.71,E2 -28369.71} C_VEL
LIN {X 0,Y 61.778,Z 613.448,A -85,B 0,C 180,E1 -28377.064,E2 -28377.064} C_VEL
LIN {X 0,Y 62.223,Z 615.409,A -85,B 0,C 180,E1 -28387.774,E2 -28387.774} C_VEL
LIN {X 0,Y 64.722,Z 616.697,A -85,B 0,C 180,E1 -28399.469,E2 -28399.469} C_VEL
LIN {X 0,Y 68.879,Z 617.034,A -85,B 0,C 180,E1 -28409.337,E2 -28409.337} C_VEL
LIN {X 0,Y 75.35,Z 616.522,A -85,B 0,C 180,E1 -28418.852,E2 -28418.852} C_VEL
LIN {X 0,Y 81.388,Z 615.43,A -85,B 0,C 180,E1 -28424.995,E2 -28424.995} C_VEL
LIN {X 0,Y 92.088,Z 612.667,A -85,B 0,C 180,E1 -28432.788,E2 -28432.788} C_VEL
LIN {X 0,Y 101.968,Z 609.314,A -85,B 0,C 180,E1 -28437.917,E2 -28437.917} C_VEL
LIN {X 0,Y 112.518,Z 604.917,A -85,B 0,C 180,E1 -28442.093,E2 -28442.093} C_VEL
LIN {X 0,Y 123.348,Z 599.568,A -85,B 0,C 180,E1 -28445.427,E2 -28445.427} C_VEL
LIN {X 0,Y 134.942,Z 592.789,A -85,B 0,C 180,E1 -28448.308,E2 -28448.308} C_VEL
LIN {X 0,Y 146.142,Z 585.059,A -85,B 0,C 180,E1 -28450.588,E2 -28450.588} C_VEL
LIN {X 0,Y 158.459,Z 575.055,A -85,B 0,C 180,E1 -28452.655,E2 -28452.655} C_VEL
LIN {X 0,Y 170.356,Z 563.507,A -85,B 0,C 180,E1 -28454.335,E2 -28454.335} C_VEL
LIN {X 0,Y 169.609,Z 564.304,A -85,B 0,C 180,E1 -28454.653,E2 -28454.653} C_VEL
LIN {X 0,Y 159.015,Z 574.757,A -85,B 0,C 180,E1 -28456.003,E2 -28456.003} C_VEL
LIN {X 0,Y 149.214,Z 583.05,A -85,B 0,C 180,E1 -28457.496,E2 -28457.496} C_VEL
LIN {X 0,Y 137.923,Z 591.353,A -85,B 0,C 180,E1 -28459.499,E2 -28459.499} C_VEL
LIN {X 0,Y 125.356,Z 599.245,A -85,B 0,C 180,E1 -28462.329,E2 -28462.329} C_VEL
LIN {X 0,Y 113.987,Z 605.319,A -85,B 0,C 180,E1 -28465.575,E2 -28465.575} C_VEL
LIN {X 0,Y 101.703,Z 610.817,A -85,B 0,C 180,E1 -28470.261,E2 -28470.261} C_VEL
LIN {X 0,Y 93.473,Z 613.841,A -85,B 0,C 180,E1 -28474.207,E2 -28474.207} C_VEL
LIN {X 0,Y 83.511,Z 616.953,A -85,B 0,C 180,E1 -28480.768,E2 -28480.768} C_VEL
LIN {X 0,Y 74.906,Z 618.951,A -85,B 0,C 180,E1 -28488.95,E2 -28488.95} C_VEL
LIN {X 0,Y 68.281,Z 619.877,A -85,B 0,C 180,E1 -28499.03,E2 -28499.03} C_VEL
LIN {X 0,Y 64.03,Z 619.784,A -85,B 0,C 180,E1 -28510.778,E2 -28510.778} C_VEL
LIN {X 0,Y 62.512,Z 618.635,A -85,B 0,C 180,E1 -28523.548,E2 -28523.548} C_VEL
LIN {X 0,Y 62.621,Z 617.605,A -85,B 0,C 180,E1 -28530.003,E2 -28530.003} C_VEL
LIN {X 0,Y 62.977,Z 614.52,A -85,B 0,C 180,E1 -28542.899,E2 -28542.899} C_VEL
LIN {X 0,Y 65.748,Z 610.096,A -85,B 0,C 180,E1 -28555.316,E2 -28555.316} C_VEL
LIN {X 0,Y 71.043,Z 604.224,A -85,B 0,C 180,E1 -28566.412,E2 -28566.412} C_VEL
LIN {X 0,Y 78.443,Z 596.742,A -85,B 0,C 180,E1 -28575.788,E2 -28575.788} C_VEL
LIN {X 0,Y 86.357,Z 588.702,A -85,B 0,C 180,E1 -28582.514,E2 -28582.514} C_VEL
LIN {X 0,Y 95.109,Z 578.959,A -85,B 0,C 180,E1 -28588.189,E2 -28588.189} C_VEL
LIN {X 0,Y 103.288,Z 569.012,A -85,B 0,C 180,E1 -28592.198,E2 -28592.198} C_VEL
LIN {X 0,Y 111.908,Z 557.181,A -85,B 0,C 180,E1 -28595.592,E2 -28595.592} C_VEL
LIN {X 0,Y 112.712,Z 555.979,A -85,B 0,C 180,E1 -28595.884,E2 -28595.884} C_VEL
LIN {X 0,Y 115.324,Z 551.37,A -85,B 0,C 180,E1 -28597.197,E2 -28597.197} C_VEL
LIN {X 0,Y 118.49,Z 543.587,A -85,B 0,C 180,E1 -28599.775,E2 -28599.775} C_VEL
LIN {X 0,Y 121.478,Z 535.538,A -85,B 0,C 180,E1 -28602.122,E2 -28602.122} C_VEL
LIN {X 0,Y 123.716,Z 530.409,A -85,B 0,C 180,E1 -28603.067,E2 -28603.067} C_VEL
LIN {X 0,Y 130.072,Z 516.267,A -85,B 0,C 180,E1 -28604.504,E2 -28604.504} C_VEL
LIN {X 0,Y 135.611,Z 500.905,A -85,B 0,C 180,E1 -28605.574,E2 -28605.574} C_VEL
LIN {X 0,Y 139.673,Z 485.717,A -85,B 0,C 180,E1 -28606.34,E2 -28606.34} C_VEL
LIN {X 0,Y 142.407,Z 470.644,A -85,B 0,C 180,E1 -28606.874,E2 -28606.874} C_VEL
LIN {X 0,Y 146.619,Z 436.496,A -85,B 0,C 180,E1 -28607.808,E2 -28607.808} C_VEL
LIN {X 0,Y 145.749,Z 433.698,A -85,B 0,C 180,E1 -28608.963,E2 -28608.963} C_VEL
LIN {X 0,Y 143.353,Z 427.584,A -85,B 0,C 180,E1 -28612.303,E2 -28612.303} C_VEL
LIN {X 0,Y 140.268,Z 420.207,A -85,B 0,C 180,E1 -28617.483,E2 -28617.483} C_VEL
LIN {X 0,Y 138.271,Z 415.617,A -85,B 0,C 180,E1 -28622.001,E2 -28622.001} C_VEL
LIN {X 0,Y 137.227,Z 412.968,A -85,B 0,C 180,E1 -28625.257,E2 -28625.257} C_VEL
LIN {X 0,Y 136.222,Z 410.226,A -85,B 0,C 180,E1 -28630.318,E2 -28630.318} C_VEL
LIN {X 0,Y 135.991,Z 410.406,A -85,B 0,C 180,E1 -28638.936,E2 -28638.936} C_VEL
LIN {X 0,Y 137.528,Z 414.584,A -85,B 0,C 180,E1 -28646.616,E2 -28646.616} C_VEL
LIN {X 0,Y 139.245,Z 418.311,A -85,B 0,C 180,E1 -28650.977,E2 -28650.977} C_VEL
LIN {X 0,Y 141.468,Z 423.211,A -85,B 0,C 180,E1 -28655.28,E2 -28655.28} C_VEL
LIN {X 0,Y 144.458,Z 430.291,A -85,B 0,C 180,E1 -28659.823,E2 -28659.823} C_VEL
LIN {X 0,Y 146.53,Z 435.674,A -85,B 0,C 180,E1 -28662.536,E2 -28662.536} C_VEL
LIN {X 0,Y 141.798,Z 472.581,A -85,B 0,C 180,E1 -28663.551,E2 -28663.551} C_VEL
LIN {X 0,Y 138.49,Z 488.227,A -85,B 0,C 180,E1 -28664.227,E2 -28664.227} C_VEL
LIN {X 0,Y 134.018,Z 503.364,A -85,B 0,C 180,E1 -28665.197,E2 -28665.197} C_VEL
LIN {X 0,Y 128.692,Z 517.316,A -85,B 0,C 180,E1 -28666.412,E2 -28666.412} C_VEL
LIN {X 0,Y 122.441,Z 530.713,A -85,B 0,C 180,E1 -28668.01,E2 -28668.01} C_VEL
LIN {X 0,Y 115.026,Z 543.868,A -85,B 0,C 180,E1 -28670.093,E2 -28670.093} C_VEL
LIN {X 0,Y 106.365,Z 556.812,A -85,B 0,C 180,E1 -28672.919,E2 -28672.919} C_VEL
LIN {X 0,Y 98.008,Z 567.668,A -85,B 0,C 180,E1 -28676.237,E2 -28676.237} C_VEL
LIN {X 0,Y 89.478,Z 577.476,A -85,B 0,C 180,E1 -28680.463,E2 -28680.463} C_VEL
LIN {X 0,Y 79.823,Z 587.396,A -85,B 0,C 180,E1 -28686.657,E2 -28686.657} C_VEL
LIN {X 0,Y 71.319,Z 595.44,A -85,B 0,C 180,E1 -28694.275,E2 -28694.275} C_VEL
LIN {X 0,Y 63.489,Z 602.703,A -85,B 0,C 180,E1 -28704.919,E2 -28704.919} C_VEL
LIN {X 0,Y 58.332,Z 607.997,A -85,B 0,C 180,E1 -28716.917,E2 -28716.917} C_VEL
LIN {X 0,Y 55.527,Z 611.473,A -85,B 0,C 180,E1 -28728.443,E2 -28728.443} C_VEL
LIN {X 0,Y 54.64,Z 614.198,A -85,B 0,C 180,E1 -28740.959,E2 -28740.959} C_VEL
LIN {X 0,Y 55.403,Z 615.638,A -85,B 0,C 180,E1 -28750.457,E2 -28750.457} C_VEL
LIN {X 0,Y 59.501,Z 617.066,A -85,B 0,C 180,E1 -28765.765,E2 -28765.765} C_VEL
LIN {X 0,Y 63.453,Z 617.256,A -85,B 0,C 180,E1 -28773.715,E2 -28773.715} C_VEL
LIN {X 0,Y 72.653,Z 616.484,A -85,B 0,C 180,E1 -28785.301,E2 -28785.301} C_VEL
LIN {X 0,Y 78.433,Z 615.492,A -85,B 0,C 180,E1 -28790.263,E2 -28790.263} C_VEL
LIN {X 0,Y 85.945,Z 613.784,A -85,B 0,C 180,E1 -28795.317,E2 -28795.317} C_VEL
LIN {X 0,Y 98.417,Z 610.021,A -85,B 0,C 180,E1 -28801.414,E2 -28801.414} C_VEL
LIN {X 0,Y 109.407,Z 605.795,A -85,B 0,C 180,E1 -28805.358,E2 -28805.358} C_VEL
LIN {X 0,Y 120.799,Z 600.541,A -85,B 0,C 180,E1 -28808.505,E2 -28808.505} C_VEL
LIN {X 0,Y 134.458,Z 592.86,A -85,B 0,C 180,E1 -28811.478,E2 -28811.478} C_VEL
LIN {X 0,Y 146.825,Z 584.478,A -85,B 0,C 180,E1 -28813.636,E2 -28813.636} C_VEL
LIN {X 0,Y 150.01,Z 582.021,A -85,B 0,C 180,E1 -28814.121,E2 -28814.121} C_VEL
LIN {X 0,Y 148.908,Z 582.908,A -85,B 0,C 180,E1 -28814.648,E2 -28814.648} C_VEL
LIN {X 0,Y 137.387,Z 591.19,A -85,B 0,C 180,E1 -28816.442,E2 -28816.442} C_VEL
LIN {X 0,Y 126.055,Z 598.181,A -85,B 0,C 180,E1 -28818.6,E2 -28818.6} C_VEL
LIN {X 0,Y 113.393,Z 604.767,A -85,B 0,C 180,E1 -28821.622,E2 -28821.622} C_VEL
LIN {X 0,Y 101.264,Z 610.013,A -85,B 0,C 180,E1 -28825.553,E2 -28825.553} C_VEL
LIN {X 0,Y 89.654,Z 614.063,A -85,B 0,C 180,E1 -28830.431,E2 -28830.431} C_VEL
LIN {X 0,Y 79.034,Z 617.002,A -85,B 0,C 180,E1 -28836.845,E2 -28836.845} C_VEL
LIN {X 0,Y 69.669,Z 618.905,A -85,B 0,C 180,E1 -28845.083,E2 -28845.083} C_VEL
LIN {X 0,Y 62.259,Z 619.707,A -85,B 0,C 180,E1 -28855.642,E2 -28855.642} C_VEL
LIN {X 0,Y 57.337,Z 619.476,A -85,B 0,C 180,E1 -28868.428,E2 -28868.428} C_VEL
LIN {X 0,Y 55.463,Z 618.205,A -85,B 0,C 180,E1 -28882.723,E2 -28882.723} C_VEL
LIN {X 0,Y 55.516,Z 617.146,A -85,B 0,C 180,E1 -28890.003,E2 -28890.003} C_VEL
LIN {X 0,Y 55.455,Z 615.714,A -85,B 0,C 180,E1 -28897.284,E2 -28897.284} C_VEL
LIN {X 0,Y 57.364,Z 611.833,A -85,B 0,C 180,E1 -28911.567,E2 -28911.567} C_VEL
LIN {X 0,Y 62.065,Z 606.545,A -85,B 0,C 180,E1 -28924.487,E2 -28924.487} C_VEL
LIN {X 0,Y 69.287,Z 599.73,A -85,B 0,C 180,E1 -28935.239,E2 -28935.239} C_VEL
LIN {X 0,Y 78.376,Z 591.191,A -85,B 0,C 180,E1 -28943.809,E2 -28943.809} C_VEL
LIN {X 0,Y 86.08,Z 583.405,A -85,B 0,C 180,E1 -28949.013,E2 -28949.013} C_VEL
LIN {X 0,Y 94.758,Z 573.789,A -85,B 0,C 180,E1 -28953.569,E2 -28953.569} C_VEL
LIN {X 0,Y 103.106,Z 563.518,A -85,B 0,C 180,E1 -28956.957,E2 -28956.957} C_VEL
LIN {X 0,Y 111.437,Z 551.787,A -85,B 0,C 180,E1 -28959.74,E2 -28959.74} C_VEL
LIN {X 0,Y 119.205,Z 539.001,A -85,B 0,C 180,E1 -28961.931,E2 -28961.931} C_VEL
LIN {X 0,Y 123.716,Z 530.409,A -85,B 0,C 180,E1 -28963.067,E2 -28963.067} C_VEL
LIN {X 0,Y 125.843,Z 525.268,A -85,B 0,C 180,E1 -28963.949,E2 -28963.949} C_VEL
LIN {X 0,Y 128.3,Z 516.651,A -85,B 0,C 180,E1 -28965.891,E2 -28965.891} C_VEL
LIN {X 0,Y 130.482,Z 507.865,A -85,B 0,C 180,E1 -28967.642,E2 -28967.642} C_VEL
LIN {X 0,Y 132.093,Z 502.329,A -85,B 0,C 180,E1 -28968.23,E2 -28968.23} C_VEL
LIN {X 0,Y 136.273,Z 487.581,A -85,B 0,C 180,E1 -28968.946,E2 -28968.946} C_VEL
LIN {X 0,Y 139.141,Z 473.232,A -85,B 0,C 180,E1 -28969.442,E2 -28969.442} C_VEL
LIN {X 0,Y 143.435,Z 439.413,A -85,B 0,C 180,E1 -28970.357,E2 -28970.357} C_VEL
LIN {X 0,Y 141.132,Z 433.154,A -85,B 0,C 180,E1 -28973.887,E2 -28973.887} C_VEL
LIN {X 0,Y 138.545,Z 426.335,A -85,B 0,C 180,E1 -28978.785,E2 -28978.785} C_VEL
LIN {X 0,Y 136.741,Z 421.859,A -85,B 0,C 180,E1 -28983.346,E2 -28983.346} C_VEL
LIN {X 0,Y 135.994,Z 419.719,A -85,B 0,C 180,E1 -28986.072,E2 -28986.072} C_VEL
LIN {X 0,Y 135.217,Z 417.297,A -85,B 0,C 180,E1 -28990.395,E2 -28990.395} C_VEL
LIN {X 0,Y 134.947,Z 417.266,A -85,B 0,C 180,E1 -28998.203,E2 -28998.203} C_VEL
LIN {X 0,Y 136.3,Z 421.459,A -85,B 0,C 180,E1 -29005.987,E2 -29005.987} C_VEL
LIN {X 0,Y 137.766,Z 424.912,A -85,B 0,C 180,E1 -29010.07,E2 -29010.07} C_VEL
LIN {X 0,Y 139.753,Z 429.694,A -85,B 0,C 180,E1 -29014.265,E2 -29014.265} C_VEL
LIN {X 0,Y 142.291,Z 436.117,A -85,B 0,C 180,E1 -29018.443,E2 -29018.443} C_VEL
LIN {X 0,Y 143.349,Z 439.095,A -85,B 0,C 180,E1 -29020.032,E2 -29020.032} C_VEL
LIN {X 0,Y 138.834,Z 473.206,A -85,B 0,C 180,E1 -29020.92,E2 -29020.92} C_VEL
LIN {X 0,Y 135.457,Z 488.729,A -85,B 0,C 180,E1 -29021.554,E2 -29021.554} C_VEL
LIN {X 0,Y 130.928,Z 503.627,A -85,B 0,C 180,E1 -29022.431,E2 -29022.431} C_VEL
LIN {X 0,Y 125.879,Z 516.637,A -85,B 0,C 180,E1 -29023.464,E2 -29023.464} C_VEL
LIN {X 0,Y 119.21,Z 530.669,A -85,B 0,C 180,E1 -29025.02,E2 -29025.02} C_VEL
LIN {X 0,Y 111.843,Z 543.436,A -85,B 0,C 180,E1 -29026.892,E2 -29026.892} C_VEL
LIN {X 0,Y 102.883,Z 556.513,A -85,B 0,C 180,E1 -29029.537,E2 -29029.537} C_VEL
LIN {X 0,Y 93.393,Z 568.331,A -85,B 0,C 180,E1 -29032.984,E2 -29032.984} C_VEL
LIN {X 0,Y 84.802,Z 577.763,A -85,B 0,C 180,E1 -29036.964,E2 -29036.964} C_VEL
LIN {X 0,Y 75.691,Z 586.629,A -85,B 0,C 180,E1 -29042.336,E2 -29042.336} C_VEL
LIN {X 0,Y 66.864,Z 594.497,A -85,B 0,C 180,E1 -29049.524,E2 -29049.524} C_VEL
LIN {X 0,Y 58.564,Z 601.55,A -85,B 0,C 180,E1 -29059.586,E2 -29059.586} C_VEL
LIN {X 0,Y 53.262,Z 606.308,A -85,B 0,C 180,E1 -29069.997,E2 -29069.997} C_VEL
LIN {X 0,Y 49.981,Z 609.617,A -85,B 0,C 180,E1 -29080.248,E2 -29080.248} C_VEL
LIN {X 0,Y 47.583,Z 613.483,A -85,B 0,C 180,E1 -29097.634,E2 -29097.634} C_VEL
LIN {X 0,Y 49.075,Z 616.05,A -85,B 0,C 180,E1 -29115.723,E2 -29115.723} C_VEL
LIN {X 0,Y 52.622,Z 617.111,A -85,B 0,C 180,E1 -29127.724,E2 -29127.724} C_VEL
LIN {X 0,Y 59.623,Z 617.454,A -85,B 0,C 180,E1 -29140.549,E2 -29140.549} C_VEL
LIN {X 0,Y 65.77,Z 617.079,A -85,B 0,C 180,E1 -29147.67,E2 -29147.67} C_VEL
LIN {X 0,Y 77.431,Z 615.34,A -85,B 0,C 180,E1 -29156.707,E2 -29156.707} C_VEL
LIN {X 0,Y 84.335,Z 613.824,A -85,B 0,C 180,E1 -29160.526,E2 -29160.526} C_VEL
LIN {X 0,Y 93.063,Z 611.449,A -85,B 0,C 180,E1 -29164.338,E2 -29164.338} C_VEL
LIN {X 0,Y 106.67,Z 606.713,A -85,B 0,C 180,E1 -29168.797,E2 -29168.797} C_VEL
LIN {X 0,Y 118.4,Z 601.57,A -85,B 0,C 180,E1 -29171.661,E2 -29171.661} C_VEL
LIN {X 0,Y 130.382,Z 595.263,A -85,B 0,C 180,E1 -29174.02,E2 -29174.02} C_VEL
LIN {X 0,Y 130.584,Z 595.162,A -85,B 0,C 180,E1 -29174.37,E2 -29174.37} C_VEL
LIN {X 0,Y 117.433,Z 602.267,A -85,B 0,C 180,E1 -29176.763,E2 -29176.763} C_VEL
LIN {X 0,Y 104.611,Z 607.993,A -85,B 0,C 180,E1 -29179.863,E2 -29179.863} C_VEL
LIN {X 0,Y 92.273,Z 612.485,A -85,B 0,C 180,E1 -29183.946,E2 -29183.946} C_VEL
LIN {X 0,Y 80.495,Z 615.811,A -85,B 0,C 180,E1 -29189.186,E2 -29189.186} C_VEL
LIN {X 0,Y 69.7,Z 618.065,A -85,B 0,C 180,E1 -29196.235,E2 -29196.235} C_VEL
LIN {X 0,Y 60.378,Z 619.306,A -85,B 0,C 180,E1 -29205.706,E2 -29205.706} C_VEL
LIN {X 0,Y 53.204,Z 619.476,A -85,B 0,C 180,E1 -29218.108,E2 -29218.108} C_VEL
LIN {X 0,Y 49.142,Z 618.591,A -85,B 0,C 180,E1 -29233.384,E2 -29233.384} C_VEL
LIN {X 0,Y 48.415,Z 617.756,A -85,B 0,C 180,E1 -29241.657,E2 -29241.657} C_VEL
LIN {X 0,Y 48.43,Z 616.635,A -85,B 0,C 180,E1 -29250.003,E2 -29250.003} C_VEL
LIN {X 0,Y 49.172,Z 613.33,A -85,B 0,C 180,E1 -29266.613,E2 -29266.613} C_VEL
LIN {X 0,Y 53.151,Z 608.636,A -85,B 0,C 180,E1 -29281.935,E2 -29281.935} C_VEL
LIN {X 0,Y 60.073,Z 602.446,A -85,B 0,C 180,E1 -29294.586,E2 -29294.586} C_VEL
LIN {X 0,Y 69.198,Z 594.607,A -85,B 0,C 180,E1 -29304.344,E2 -29304.344} C_VEL
LIN {X 0,Y 78.429,Z 586.207,A -85,B 0,C 180,E1 -29310.893,E2 -29310.893} C_VEL
LIN {X 0,Y 87.946,Z 576.452,A -85,B 0,C 180,E1 -29315.988,E2 -29315.988} C_VEL
LIN {X 0,Y 97.41,Z 565.602,A -85,B 0,C 180,E1 -29319.709,E2 -29319.709} C_VEL
LIN {X 0,Y 106.759,Z 553.16,A -85,B 0,C 180,E1 -29322.66,E2 -29322.66} C_VEL
LIN {X 0,Y 114.743,Z 540.694,A -85,B 0,C 180,E1 -29324.728,E2 -29324.728} C_VEL
LIN {X 0,Y 122.032,Z 527.093,A -85,B 0,C 180,E1 -29326.374,E2 -29326.374} C_VEL
LIN {X 0,Y 128.105,Z 513.302,A -85,B 0,C 180,E1 -29327.573,E2 -29327.573} C_VEL
LIN {X 0,Y 132.093,Z 502.329,A -85,B 0,C 180,E1 -29328.23,E2 -29328.23} C_VEL
LIN {X 0,Y 133.599,Z 496.748,A -85,B 0,C 180,E1 -29328.771,E2 -29328.771} C_VEL
LIN {X 0,Y 134.959,Z 487.596,A -85,B 0,C 180,E1 -29330.31,E2 -29330.31} C_VEL
LIN {X 0,Y 135.928,Z 478.315,A -85,B 0,C 180,E1 -29331.761,E2 -29331.761} C_VEL
LIN {X 0,Y 136.656,Z 472.526,A -85,B 0,C 180,E1 -29332.203,E2 -29332.203} C_VEL
LIN {X 0,Y 140.54,Z 443.051,A -85,B 0,C 180,E1 -29332.892,E2 -29332.892} C_VEL
LIN {X 0,Y 138.336,Z 436.779,A -85,B 0,C 180,E1 -29336.803,E2 -29336.803} C_VEL
LIN {X 0,Y 136.693,Z 432.097,A -85,B 0,C 180,E1 -29340.556,E2 -29340.556} C_VEL
LIN {X 0,Y 135.352,Z 428.264,A -85,B 0,C 180,E1 -29344.497,E2 -29344.497} C_VEL
LIN {X 0,Y 134.785,Z 426.425,A -85,B 0,C 180,E1 -29346.935,E2 -29346.935} C_VEL
LIN {X 0,Y 134.165,Z 424.306,A -85,B 0,C 180,E1 -29350.799,E2 -29350.799} C_VEL
LIN {X 0,Y 133.935,Z 424.38,A -85,B 0,C 180,E1 -29358.019,E2 -29358.019} C_VEL
LIN {X 0,Y 135.064,Z 428.237,A -85,B 0,C 180,E1 -29365.242,E2 -29365.242} C_VEL
LIN {X 0,Y 136.266,Z 431.404,A -85,B 0,C 180,E1 -29369.022,E2 -29369.022} C_VEL
LIN {X 0,Y 137.981,Z 435.86,A -85,B 0,C 180,E1 -29373.007,E2 -29373.007} C_VEL
LIN {X 0,Y 140.207,Z 442.05,A -85,B 0,C 180,E1 -29377.103,E2 -29377.103} C_VEL
LIN {X 0,Y 140.398,Z 442.607,A -85,B 0,C 180,E1 -29377.416,E2 -29377.416} C_VEL
LIN {X 0,Y 136.242,Z 473.279,A -85,B 0,C 180,E1 -29378.167,E2 -29378.167} C_VEL
LIN {X 0,Y 132.889,Z 488.508,A -85,B 0,C 180,E1 -29378.733,E2 -29378.733} C_VEL
LIN {X 0,Y 128.164,Z 503.769,A -85,B 0,C 180,E1 -29379.544,E2 -29379.544} C_VEL
LIN {X 0,Y 122.598,Z 517.699,A -85,B 0,C 180,E1 -29380.574,E2 -29380.574} C_VEL
LIN {X 0,Y 115.419,Z 532.121,A -85,B 0,C 180,E1 -29382.043,E2 -29382.043} C_VEL
LIN {X 0,Y 107.306,Z 545.505,A -85,B 0,C 180,E1 -29383.908,E2 -29383.908} C_VEL
LIN {X 0,Y 99.248,Z 556.811,A -85,B 0,C 180,E1 -29386.082,E2 -29386.082} C_VEL
LIN {X 0,Y 89.125,Z 568.916,A -85,B 0,C 180,E1 -29389.415,E2 -29389.415} C_VEL
LIN {X 0,Y 79.487,Z 578.948,A -85,B 0,C 180,E1 -29393.552,E2 -29393.552} C_VEL
LIN {X 0,Y 69.077,Z 588.383,A -85,B 0,C 180,E1 -29399.42,E2 -29399.42} C_VEL
LIN {X 0,Y 60.329,Z 595.58,A -85,B 0,C 180,E1 -29406.449,E2 -29406.449} C_VEL
LIN {X 0,Y 51.549,Z 602.423,A -85,B 0,C 180,E1 -29417.25,E2 -29417.25} C_VEL
LIN {X 0,Y 45.505,Z 607.351,A -85,B 0,C 180,E1 -29429.996,E2 -29429.996} C_VEL
LIN {X 0,Y 41.711,Z 611.105,A -85,B 0,C 180,E1 -29444.63,E2 -29444.63} C_VEL
LIN {X 0,Y 40.445,Z 613.985,A -85,B 0,C 180,E1 -29461.414,E2 -29461.414} C_VEL
LIN {X 0,Y 42.3,Z 616.078,A -85,B 0,C 180,E1 -29478.372,E2 -29478.372} C_VEL
LIN {X 0,Y 47.172,Z 617.319,A -85,B 0,C 180,E1 -29493.468,E2 -29493.468} C_VEL
LIN {X 0,Y 57.311,Z 617.646,A -85,B 0,C 180,E1 -29508.8,E2 -29508.8} C_VEL
LIN {X 0,Y 70.281,Z 616.409,A -85,B 0,C 180,E1 -29519.286,E2 -29519.286} C_VEL
LIN {X 0,Y 81.232,Z 614.357,A -85,B 0,C 180,E1 -29524.971,E2 -29524.971} C_VEL
LIN {X 0,Y 92.538,Z 611.476,A -85,B 0,C 180,E1 -29529.155,E2 -29529.155} C_VEL
LIN {X 0,Y 104.991,Z 607.332,A -85,B 0,C 180,E1 -29532.564,E2 -29532.564} C_VEL
LIN {X 0,Y 110.418,Z 605.174,A -85,B 0,C 180,E1 -29533.766,E2 -29533.766} C_VEL
LIN {X 0,Y 108.967,Z 605.813,A -85,B 0,C 180,E1 -29534.67,E2 -29534.67} C_VEL
LIN {X 0,Y 95.974,Z 610.729,A -85,B 0,C 180,E1 -29537.84,E2 -29537.84} C_VEL
LIN {X 0,Y 83.339,Z 614.505,A -85,B 0,C 180,E1 -29541.94,E2 -29541.94} C_VEL
LIN {X 0,Y 71.381,Z 617.133,A -85,B 0,C 180,E1 -29547.617,E2 -29547.617} C_VEL
LIN {X 0,Y 59.461,Z 618.813,A -85,B 0,C 180,E1 -29556.239,E2 -29556.239} C_VEL
LIN {X 0,Y 51.072,Z 619.309,A -85,B 0,C 180,E1 -29566.53,E2 -29566.53} C_VEL
LIN {X 0,Y 44.355,Z 618.85,A -85,B 0,C 180,E1 -29581.623,E2 -29581.623} C_VEL
LIN {X 0,Y 41.382,Z 617.299,A -85,B 0,C 180,E1 -29600.226,E2 -29600.226} C_VEL
LIN {X 0,Y 41.325,Z 616.106,A -85,B 0,C 180,E1 -29610.004,E2 -29610.004} C_VEL
LIN {X 0,Y 42.399,Z 612.647,A -85,B 0,C 180,E1 -29629.364,E2 -29629.364} C_VEL
LIN {X 0,Y 47.225,Z 607.801,A -85,B 0,C 180,E1 -29646.536,E2 -29646.536} C_VEL
LIN {X 0,Y 55.196,Z 601.449,A -85,B 0,C 180,E1 -29659.818,E2 -29659.818} C_VEL
LIN {X 0,Y 65.253,Z 593.413,A -85,B 0,C 180,E1 -29669.503,E2 -29669.503} C_VEL
LIN {X 0,Y 75.189,Z 584.826,A -85,B 0,C 180,E1 -29675.695,E2 -29675.695} C_VEL
LIN {X 0,Y 84.851,Z 575.298,A -85,B 0,C 180,E1 -29680.25,E2 -29680.25} C_VEL
LIN {X 0,Y 95.154,Z 563.739,A -85,B 0,C 180,E1 -29683.777,E2 -29683.777} C_VEL
LIN {X 0,Y 104.032,Z 552.141,A -85,B 0,C 180,E1 -29686.198,E2 -29686.198} C_VEL
LIN {X 0,Y 112.236,Z 539.519,A -85,B 0,C 180,E1 -29688.072,E2 -29688.072} C_VEL
LIN {X 0,Y 119.711,Z 525.71,A -85,B 0,C 180,E1 -29689.534,E2 -29689.534} C_VEL
LIN {X 0,Y 126.174,Z 510.967,A -85,B 0,C 180,E1 -29690.646,E2 -29690.646} C_VEL
LIN {X 0,Y 131.284,Z 496.238,A -85,B 0,C 180,E1 -29691.371,E2 -29691.371} C_VEL
LIN {X 0,Y 135.069,Z 481.31,A -85,B 0,C 180,E1 -29691.932,E2 -29691.932} C_VEL
LIN {X 0,Y 136.656,Z 472.526,A -85,B 0,C 180,E1 -29692.203,E2 -29692.203} C_VEL
LIN {X 0,Y 136.998,Z 468.652,A -85,B 0,C 180,E1 -29692.576,E2 -29692.576} C_VEL
LIN {X 0,Y 136.713,Z 456.57,A -85,B 0,C 180,E1 -29695.095,E2 -29695.095} C_VEL
LIN {X 0,Y 137.012,Z 452.686,A -85,B 0,C 180,E1 -29695.444,E2 -29695.444} C_VEL
LIN {X 0,Y 137.764,Z 446.828,A -85,B 0,C 180,E1 -29695.58,E2 -29695.58} C_VEL
LIN {X 0,Y 135.924,Z 440.669,A -85,B 0,C 180,E1 -29699.748,E2 -29699.748} C_VEL
LIN {X 0,Y 134.165,Z 435.201,A -85,B 0,C 180,E1 -29705.043,E2 -29705.043} C_VEL
LIN {X 0,Y 133.605,Z 433.146,A -85,B 0,C 180,E1 -29707.797,E2 -29707.797} C_VEL
LIN {X 0,Y 133.106,Z 431.309,A -85,B 0,C 180,E1 -29711.309,E2 -29711.309} C_VEL
LIN {X 0,Y 132.925,Z 431.518,A -85,B 0,C 180,E1 -29717.881,E2 -29717.881} C_VEL
LIN {X 0,Y 133.85,Z 435.003,A -85,B 0,C 180,E1 -29724.472,E2 -29724.472} C_VEL
LIN {X 0,Y 134.936,Z 438.225,A -85,B 0,C 180,E1 -29728.311,E2 -29728.311} C_VEL
LIN {X 0,Y 136.633,Z 443.148,A -85,B 0,C 180,E1 -29732.553,E2 -29732.553} C_VEL
LIN {X 0,Y 137.671,Z 446.529,A -85,B 0,C 180,E1 -29734.768,E2 -29734.768} C_VEL
LIN {X 0,Y 133.861,Z 473.629,A -85,B 0,C 180,E1 -29735.34,E2 -29735.34} C_VEL
LIN {X 0,Y 130.289,Z 489.348,A -85,B 0,C 180,E1 -29735.861,E2 -29735.861} C_VEL
LIN {X 0,Y 125.74,Z 503.745,A -85,B 0,C 180,E1 -29736.538,E2 -29736.538} C_VEL
LIN {X 0,Y 120.481,Z 516.783,A -85,B 0,C 180,E1 -29737.365,E2 -29737.365} C_VEL
LIN {X 0,Y 113.702,Z 530.457,A -85,B 0,C 180,E1 -29738.587,E2 -29738.587} C_VEL
LIN {X 0,Y 105.726,Z 543.66,A -85,B 0,C 180,E1 -29740.141,E2 -29740.141} C_VEL
LIN {X 0,Y 96.231,Z 556.768,A -85,B 0,C 180,E1 -29742.314,E2 -29742.314} C_VEL
LIN {X 0,Y 86.909,Z 567.693,A -85,B 0,C 180,E1 -29744.96,E2 -29744.96} C_VEL
LIN {X 0,Y 76.983,Z 577.749,A -85,B 0,C 180,E1 -29748.555,E2 -29748.555} C_VEL
LIN {X 0,Y 65.774,Z 587.591,A -85,B 0,C 180,E1 -29754.005,E2 -29754.005} C_VEL
LIN {X 0,Y 55.404,Z 595.592,A -85,B 0,C 180,E1 -29761.385,E2 -29761.385} C_VEL
LIN {X 0,Y 45.91,Z 602.349,A -85,B 0,C 180,E1 -29772.168,E2 -29772.168} C_VEL
LIN {X 0,Y 39.463,Z 607.014,A -85,B 0,C 180,E1 -29784.887,E2 -29784.887} C_VEL
LIN {X 0,Y 34.904,Z 610.873,A -85,B 0,C 180,E1 -29801.611,E2 -29801.611} C_VEL
LIN {X 0,Y 33.36,Z 613.96,A -85,B 0,C 180,E1 -29822.613,E2 -29822.613} C_VEL
LIN {X 0,Y 36.175,Z 616.279,A -85,B 0,C 180,E1 -29844.373,E2 -29844.373} C_VEL
LIN {X 0,Y 43.965,Z 617.705,A -85,B 0,C 180,E1 -29863.543,E2 -29863.543} C_VEL
LIN {X 0,Y 56.27,Z 617.783,A -85,B 0,C 180,E1 -29877.576,E2 -29877.576} C_VEL
LIN {X 0,Y 70.72,Z 616.297,A -85,B 0,C 180,E1 -29886.427,E2 -29886.427} C_VEL
LIN {X 0,Y 79.836,Z 614.657,A -85,B 0,C 180,E1 -29890.149,E2 -29890.149} C_VEL
LIN {X 0,Y 90.626,Z 612.104,A -85,B 0,C 180,E1 -29893.46,E2 -29893.46} C_VEL
LIN {X 0,Y 87.463,Z 613.008,A -85,B 0,C 180,E1 -29895.38,E2 -29895.38} C_VEL
LIN {X 0,Y 74.571,Z 616.071,A -85,B 0,C 180,E1 -29899.542,E2 -29899.542} C_VEL
LIN {X 0,Y 62.324,Z 618.047,A -85,B 0,C 180,E1 -29905.569,E2 -29905.569} C_VEL
LIN {X 0,Y 51.104,Z 618.971,A -85,B 0,C 180,E1 -29914.405,E2 -29914.405} C_VEL
LIN {X 0,Y 41.764,Z 618.908,A -85,B 0,C 180,E1 -29927.698,E2 -29927.698} C_VEL
LIN {X 0,Y 35.711,Z 617.816,A -85,B 0,C 180,E1 -29946.826,E2 -29946.826} C_VEL
LIN {X 0,Y 34.399,Z 616.841,A -85,B 0,C 180,E1 -29958.216,E2 -29958.216} C_VEL
LIN {X 0,Y 34.237,Z 615.578,A -85,B 0,C 180,E1 -29970.005,E2 -29970.005} C_VEL
LIN {X 0,Y 35.738,Z 611.963,A -85,B 0,C 180,E1 -29993.165,E2 -29993.165} C_VEL
LIN {X 0,Y 41.689,Z 606.952,A -85,B 0,C 180,E1 -30012.406,E2 -30012.406} C_VEL
LIN {X 0,Y 50.853,Z 600.422,A -85,B 0,C 180,E1 -30026.021,E2 -30026.021} C_VEL
LIN {X 0,Y 61.915,Z 592.195,A -85,B 0,C 180,E1 -30035.246,E2 -30035.246} C_VEL
LIN {X 0,Y 72.51,Z 583.385,A -85,B 0,C 180,E1 -30040.915,E2 -30040.915} C_VEL
LIN {X 0,Y 83.309,Z 572.99,A -85,B 0,C 180,E1 -30045.145,E2 -30045.145} C_VEL
LIN {X 0,Y 93.401,Z 561.772,A -85,B 0,C 180,E1 -30048.013,E2 -30048.013} C_VEL
LIN {X 0,Y 102.558,Z 549.827,A -85,B 0,C 180,E1 -30050.091,E2 -30050.091} C_VEL
LIN {X 0,Y 110.978,Z 536.766,A -85,B 0,C 180,E1 -30051.69,E2 -30051.69} C_VEL
LIN {X 0,Y 118.617,Z 522.361,A -85,B 0,C 180,E1 -30052.945,E2 -30052.945} C_VEL
LIN {X 0,Y 124.595,Z 508.395,A -85,B 0,C 180,E1 -30053.799,E2 -30053.799} C_VEL
LIN {X 0,Y 129.478,Z 493.852,A -85,B 0,C 180,E1 -30054.41,E2 -30054.41} C_VEL
LIN {X 0,Y 133.205,Z 478.623,A -85,B 0,C 180,E1 -30054.855,E2 -30054.855} C_VEL
LIN {X 0,Y 136.29,Z 458.265,A -85,B 0,C 180,E1 -30055.32,E2 -30055.32} C_VEL
LIN {X 0,Y 137.012,Z 452.686,A -85,B 0,C 180,E1 -30055.444,E2 -30055.444} C_VEL
LIN {X 0,Y 137.065,Z 450.52,A -85,B 0,C 180,E1 -30055.798,E2 -30055.798} C_VEL
LIN {X 0,Y 136.682,Z 448.494,A -85,B 0,C 180,E1 -30056.747,E2 -30056.747} C_VEL
LIN {X 0,Y 135.772,Z 446.826,A -85,B 0,C 180,E1 -30058.495,E2 -30058.495} C_VEL
LIN {X 0,Y 133.671,Z 444.693,A -85,B 0,C 180,E1 -30062.963,E2 -30062.963} C_VEL
LIN {X 0,Y 133.477,Z 444.146,A -85,B 0,C 180,E1 -30063.581,E2 -30063.581} C_VEL
LIN {X 0,Y 132.591,Z 440.343,A -85,B 0,C 180,E1 -30067.8,E2 -30067.8} C_VEL
LIN {X 0,Y 132.105,Z 438.376,A -85,B 0,C 180,E1 -30071.396,E2 -30071.396} C_VEL
LIN {X 0,Y 131.921,Z 438.402,A -85,B 0,C 180,E1 -30077.311,E2 -30077.311} C_VEL
LIN {X 0,Y 132.662,Z 441.785,A -85,B 0,C 180,E1 -30083.699,E2 -30083.699} C_VEL
LIN {X 0,Y 133.53,Z 444.746,A -85,B 0,C 180,E1 -30087.271,E2 -30087.271} C_VEL
LIN {X 0,Y 134.917,Z 449.162,A -85,B 0,C 180,E1 -30091.148,E2 -30091.148} C_VEL
LIN {X 0,Y 135.221,Z 450.236,A -85,B 0,C 180,E1 -30091.923,E2 -30091.923} C_VEL
LIN {X 0,Y 131.638,Z 474.889,A -85,B 0,C 180,E1 -30092.444,E2 -30092.444} C_VEL
LIN {X 0,Y 127.964,Z 490.405,A -85,B 0,C 180,E1 -30092.884,E2 -30092.884} C_VEL
LIN {X 0,Y 123.204,Z 504.918,A -85,B 0,C 180,E1 -30093.46,E2 -30093.46} C_VEL
LIN {X 0,Y 117.019,Z 519.566,A -85,B 0,C 180,E1 -30094.329,E2 -30094.329} C_VEL
LIN {X 0,Y 109.884,Z 533.134,A -85,B 0,C 180,E1 -30095.397,E2 -30095.397} C_VEL
LIN {X 0,Y 101.917,Z 545.67,A -85,B 0,C 180,E1 -30096.712,E2 -30096.712} C_VEL
LIN {X 0,Y 93.114,Z 557.379,A -85,B 0,C 180,E1 -30098.456,E2 -30098.456} C_VEL
LIN {X 0,Y 83.497,Z 568.261,A -85,B 0,C 180,E1 -30100.751,E2 -30100.751} C_VEL
LIN {X 0,Y 73.224,Z 578.247,A -85,B 0,C 180,E1 -30103.957,E2 -30103.957} C_VEL
LIN {X 0,Y 61.464,Z 588.034,A -85,B 0,C 180,E1 -30108.89,E2 -30108.89} C_VEL
LIN {X 0,Y 50.243,Z 596.1,A -85,B 0,C 180,E1 -30115.974,E2 -30115.974} C_VEL
LIN {X 0,Y 41.408,Z 601.817,A -85,B 0,C 180,E1 -30124.889,E2 -30124.889} C_VEL
LIN {X 0,Y 33.835,Z 606.644,A -85,B 0,C 180,E1 -30138.007,E2 -30138.007} C_VEL
LIN {X 0,Y 28.299,Z 610.521,A -85,B 0,C 180,E1 -30156.805,E2 -30156.805} C_VEL
LIN {X 0,Y 26.407,Z 614.176,A -85,B 0,C 180,E1 -30187.063,E2 -30187.063} C_VEL
LIN {X 0,Y 31.145,Z 616.612,A -85,B 0,C 180,E1 -30214.491,E2 -30214.491} C_VEL
LIN {X 0,Y 38.221,Z 617.721,A -85,B 0,C 180,E1 -30229.422,E2 -30229.422} C_VEL
LIN {X 0,Y 49.209,Z 618.133,A -85,B 0,C 180,E1 -30241.49,E2 -30241.49} C_VEL
LIN {X 0,Y 64.29,Z 617.219,A -85,B 0,C 180,E1 -30250.329,E2 -30250.329} C_VEL
LIN {X 0,Y 72.235,Z 616.169,A -85,B 0,C 180,E1 -30253.376,E2 -30253.376} C_VEL
LIN {X 0,Y 72.492,Z 616.156,A -85,B 0,C 180,E1 -30254.204,E2 -30254.204} C_VEL
LIN {X 0,Y 59.587,Z 618.016,A -85,B 0,C 180,E1 -30259.354,E2 -30259.354} C_VEL
LIN {X 0,Y 47.419,Z 618.806,A -85,B 0,C 180,E1 -30267.228,E2 -30267.228} C_VEL
LIN {X 0,Y 36.799,Z 618.588,A -85,B 0,C 180,E1 -30280.196,E2 -30280.196} C_VEL
LIN {X 0,Y 29.287,Z 617.367,A -85,B 0,C 180,E1 -30301.326,E2 -30301.326} C_VEL
LIN {X 0,Y 27.488,Z 616.361,A -85,B 0,C 180,E1 -30315.193,E2 -30315.193} C_VEL
LIN {X 0,Y 27.123,Z 615.029,A -85,B 0,C 180,E1 -30330.006,E2 -30330.006} C_VEL
LIN {X 0,Y 29.313,Z 611.261,A -85,B 0,C 180,E1 -30358.659,E2 -30358.659} C_VEL
LIN {X 0,Y 36.701,Z 606.083,A -85,B 0,C 180,E1 -30379.998,E2 -30379.998} C_VEL
LIN {X 0,Y 47.931,Z 598.928,A -85,B 0,C 180,E1 -30393.888,E2 -30393.888} C_VEL
LIN {X 0,Y 59.27,Z 590.974,A -85,B 0,C 180,E1 -30401.556,E2 -30401.556} C_VEL
LIN {X 0,Y 70.48,Z 581.946,A -85,B 0,C 180,E1 -30406.472,E2 -30406.472} C_VEL
LIN {X 0,Y 80.972,Z 572.09,A -85,B 0,C 180,E1 -30409.822,E2 -30409.822} C_VEL
LIN {X 0,Y 90.478,Z 561.786,A -85,B 0,C 180,E1 -30412.046,E2 -30412.046} C_VEL
LIN {X 0,Y 99.855,Z 549.885,A -85,B 0,C 180,E1 -30413.803,E2 -30413.803} C_VEL
LIN {X 0,Y 108.444,Z 536.874,A -85,B 0,C 180,E1 -30415.154,E2 -30415.154} C_VEL
LIN {X 0,Y 116.04,Z 522.896,A -85,B 0,C 180,E1 -30416.187,E2 -30416.187} C_VEL
LIN {X 0,Y 122.289,Z 508.666,A -85,B 0,C 180,E1 -30416.916,E2 -30416.916} C_VEL
LIN {X 0,Y 127.274,Z 494.147,A -85,B 0,C 180,E1 -30417.423,E2 -30417.423} C_VEL
LIN {X 0,Y 131.208,Z 478.374,A -85,B 0,C 180,E1 -30417.798,E2 -30417.798} C_VEL
LIN {X 0,Y 134.256,Z 458.595,A -85,B 0,C 180,E1 -30418.205,E2 -30418.205} C_VEL
LIN {X 0,Y 135.299,Z 450.558,A -85,B 0,C 180,E1 -30418.39,E2 -30418.39} C_VEL
LIN {X 0,Y 133.852,Z 445.305,A -85,B 0,C 180,E1 -30422.385,E2 -30422.385} C_VEL
LIN {X 0,Y 133.477,Z 444.146,A -85,B 0,C 180,E1 -30423.581,E2 -30423.581} C_VEL
LIN {X 0,Y 132.974,Z 443.241,A -85,B 0,C 180,E1 -30425.206,E2 -30425.206} C_VEL
LIN {X 0,Y 132.419,Z 443.31,A -85,B 0,C 180,E1 -30426.903,E2 -30426.903} C_VEL
LIN {X 0,Y 131.048,Z 445.281,A -85,B 0,C 180,E1 -30432.145,E2 -30432.145} C_VEL
LIN {X 0,Y 130.984,Z 445.324,A -85,B 0,C 180,E1 -30432.743,E2 -30432.743} C_VEL
LIN {X 0,Y 130.918,Z 445.417,A -85,B 0,C 180,E1 -30436.888,E2 -30436.888} C_VEL
LIN {X 0,Y 131.479,Z 448.555,A -85,B 0,C 180,E1 -30442.917,E2 -30442.917} C_VEL
LIN {X 0,Y 132.373,Z 451.979,A -85,B 0,C 180,E1 -30446.967,E2 -30446.967} C_VEL
LIN {X 0,Y 132.997,Z 454.314,A -85,B 0,C 180,E1 -30449.03,E2 -30449.03} C_VEL
LIN {X 0,Y 129.89,Z 475.093,A -85,B 0,C 180,E1 -30449.437,E2 -30449.437} C_VEL
LIN {X 0,Y 126.116,Z 490.756,A -85,B 0,C 180,E1 -30449.792,E2 -30449.792} C_VEL
LIN {X 0,Y 121.059,Z 505.823,A -85,B 0,C 180,E1 -30450.281,E2 -30450.281} C_VEL
LIN {X 0,Y 114.787,Z 520.309,A -85,B 0,C 180,E1 -30450.999,E2 -30450.999} C_VEL
LIN {X 0,Y 107.563,Z 533.718,A -85,B 0,C 180,E1 -30451.853,E2 -30451.853} C_VEL
LIN {X 0,Y 99.431,Z 546.219,A -85,B 0,C 180,E1 -30452.928,E2 -30452.928} C_VEL
LIN {X 0,Y 90.447,Z 557.866,A -85,B 0,C 180,E1 -30454.35,E2 -30454.35} C_VEL
LIN {X 0,Y 80.551,Z 568.747,A -85,B 0,C 180,E1 -30456.225,E2 -30456.225} C_VEL
LIN {X 0,Y 69.989,Z 578.67,A -85,B 0,C 180,E1 -30458.899,E2 -30458.899} C_VEL
LIN {X 0,Y 57.707,Z 588.421,A -85,B 0,C 180,E1 -30463.05,E2 -30463.05} C_VEL
LIN {X 0,Y 46.775,Z 595.829,A -85,B 0,C 180,E1 -30468.676,E2 -30468.676} C_VEL
LIN {X 0,Y 34.639,Z 603.034,A -85,B 0,C 180,E1 -30479.516,E2 -30479.516} C_VEL
LIN {X 0,Y 26.281,Z 607.648,A -85,B 0,C 180,E1 -30494.484,E2 -30494.484} C_VEL
LIN {X 0,Y 21.123,Z 610.788,A -85,B 0,C 180,E1 -30513.979,E2 -30513.979} C_VEL
LIN {X 0,Y 19.761,Z 614.439,A -85,B 0,C 180,E1 -30555.328,E2 -30555.328} C_VEL
LIN {X 0,Y 25.871,Z 616.662,A -85,B 0,C 180,E1 -30584.264,E2 -30584.264} C_VEL
LIN {X 0,Y 35.225,Z 617.913,A -85,B 0,C 180,E1 -30600.019,E2 -30600.019} C_VEL
LIN {X 0,Y 50.199,Z 618.329,A -85,B 0,C 180,E1 -30611.493,E2 -30611.493} C_VEL
LIN {X 0,Y 52.938,Z 618.269,A -85,B 0,C 180,E1 -30612.844,E2 -30612.844} C_VEL
LIN {X 0,Y 51.02,Z 618.41,A -85,B 0,C 180,E1 -30615.383,E2 -30615.383} C_VEL
LIN {X 0,Y 38.426,Z 618.573,A -85,B 0,C 180,E1 -30623.881,E2 -30623.881} C_VEL
LIN {X 0,Y 27.439,Z 617.698,A -85,B 0,C 180,E1 -30639.8,E2 -30639.8} C_VEL
LIN {X 0,Y 20.684,Z 615.813,A -85,B 0,C 180,E1 -30670.146,E2 -30670.146} C_VEL
LIN {X 0,Y 20.011,Z 614.441,A -85,B 0,C 180,E1 -30690.008,E2 -30690.008} C_VEL
LIN {X 0,Y 23.293,Z 610.541,A -85,B 0,C 180,E1 -30727.125,E2 -30727.125} C_VEL
LIN {X 0,Y 32.556,Z 605.187,A -85,B 0,C 180,E1 -30749.721,E2 -30749.721} C_VEL
LIN {X 0,Y 44.454,Z 598.301,A -85,B 0,C 180,E1 -30761.552,E2 -30761.552} C_VEL
LIN {X 0,Y 55.752,Z 590.826,A -85,B 0,C 180,E1 -30767.684,E2 -30767.684} C_VEL
LIN {X 0,Y 67.457,Z 581.811,A -85,B 0,C 180,E1 -30771.798,E2 -30771.798} C_VEL
LIN {X 0,Y 77.677,Z 572.57,A -85,B 0,C 180,E1 -30774.418,E2 -30774.418} C_VEL
LIN {X 0,Y 88.032,Z 561.695,A -85,B 0,C 180,E1 -30776.323,E2 -30776.323} C_VEL
LIN {X 0,Y 97.592,Z 549.825,A -85,B 0,C 180,E1 -30777.712,E2 -30777.712} C_VEL
LIN {X 0,Y 106.324,Z 536.859,A -85,B 0,C 180,E1 -30778.767,E2 -30778.767} C_VEL
LIN {X 0,Y 113.888,Z 523.225,A -85,B 0,C 180,E1 -30779.559,E2 -30779.559} C_VEL
LIN {X 0,Y 120.355,Z 508.791,A -85,B 0,C 180,E1 -30780.134,E2 -30780.134} C_VEL
LIN {X 0,Y 125.411,Z 494.344,A -85,B 0,C 180,E1 -30780.517,E2 -30780.517} C_VEL
LIN {X 0,Y 129.498,Z 478.196,A -85,B 0,C 180,E1 -30780.82,E2 -30780.82} C_VEL
LIN {X 0,Y 132.765,Z 457.201,A -85,B 0,C 180,E1 -30781.164,E2 -30781.164} C_VEL
LIN {X 0,Y 133.09,Z 454.555,A -85,B 0,C 180,E1 -30781.266,E2 -30781.266} C_VEL
LIN {X 0,Y 132.133,Z 450.692,A -85,B 0,C 180,E1 -30784.62,E2 -30784.62} C_VEL
LIN {X 0,Y 131.41,Z 447.025,A -85,B 0,C 180,E1 -30788.711,E2 -30788.711} C_VEL
LIN {X 0,Y 131.093,Z 445.523,A -85,B 0,C 180,E1 -30791.485,E2 -30791.485} C_VEL
LIN {X 0,Y 130.984,Z 445.324,A -85,B 0,C 180,E1 -30792.743,E2 -30792.743} C_VEL
LIN {X 0,Y 130.84,Z 445.745,A -85,B 0,C 180,E1 -30794.45,E2 -30794.45} C_VEL
LIN {X 0,Y 130.629,Z 447.602,A -85,B 0,C 180,E1 -30796.914,E2 -30796.914} C_VEL
LIN {X 0,Y 130.481,Z 450.35,A -85,B 0,C 180,E1 -30799.243,E2 -30799.243} C_VEL
LIN {X 0,Y 130.647,Z 456.525,A -85,B 0,C 180,E1 -30803.902,E2 -30803.902} C_VEL
LIN {X 0,Y 130.942,Z 458.165,A -85,B 0,C 180,E1 -30805.534,E2 -30805.534} C_VEL
LIN {X 0,Y 131.064,Z 458.659,A -85,B 0,C 180,E1 -30806.056,E2 -30806.056} C_VEL
LIN {X 0,Y 128.232,Z 476.507,A -85,B 0,C 180,E1 -30806.37,E2 -30806.37} C_VEL
LIN {X 0,Y 124.336,Z 492.082,A -85,B 0,C 180,E1 -30806.646,E2 -30806.646} C_VEL
LIN {X 0,Y 119.303,Z 506.675,A -85,B 0,C 180,E1 -30807.001,E2 -30807.001} C_VEL
LIN {X 0,Y 112.964,Z 521.013,A -85,B 0,C 180,E1 -30807.556,E2 -30807.556} C_VEL
LIN {X 0,Y 105.649,Z 534.329,A -85,B 0,C 180,E1 -30808.185,E2 -30808.185} C_VEL
LIN {X 0,Y 96.477,Z 548.012,A -85,B 0,C 180,E1 -30809.053,E2 -30809.053} C_VEL
LIN {X 0,Y 86.425,Z 560.439,A -85,B 0,C 180,E1 -30810.228,E2 -30810.228} C_VEL
LIN {X 0,Y 76.393,Z 570.897,A -85,B 0,C 180,E1 -30811.68,E2 -30811.68} C_VEL
LIN {X 0,Y 65.789,Z 580.342,A -85,B 0,C 180,E1 -30813.702,E2 -30813.702} C_VEL
LIN {X 0,Y 54.638,Z 588.8,A -85,B 0,C 180,E1 -30816.49,E2 -30816.49} C_VEL
LIN {X 0,Y 42.857,Z 596.365,A -85,B 0,C 180,E1 -30820.97,E2 -30820.97} C_VEL
LIN {X 0,Y 31.672,Z 602.474,A -85,B 0,C 180,E1 -30828.259,E2 -30828.259} C_VEL
LIN {X 0,Y 21.86,Z 607.249,A -85,B 0,C 180,E1 -30841.159,E2 -30841.159} C_VEL
LIN {X 0,Y 13.78,Z 611.178,A -85,B 0,C 180,E1 -30869.988,E2 -30869.988} C_VEL
LIN {X 0,Y 13.636,Z 614.56,A -85,B 0,C 180,E1 -30929.033,E2 -30929.033} C_VEL
LIN {X 0,Y 22.686,Z 616.849,A -85,B 0,C 180,E1 -30960.029,E2 -30960.029} C_VEL
LIN {X 0,Y 33.644,Z 618.106,A -85,B 0,C 180,E1 -30972.078,E2 -30972.078} C_VEL
LIN {X 0,Y 29.65,Z 617.931,A -85,B 0,C 180,E1 -30978.555,E2 -30978.555} C_VEL
LIN {X 0,Y 18.126,Z 616.397,A -85,B 0,C 180,E1 -30999.17,E2 -30999.17} C_VEL
LIN {X 0,Y 14.205,Z 615.244,A -85,B 0,C 180,E1 -31020.36,E2 -31020.36} C_VEL
LIN {X 0,Y 12.913,Z 613.798,A -85,B 0,C 180,E1 -31050.012,E2 -31050.012} C_VEL
LIN {X 0,Y 15.899,Z 610.889,A -85,B 0,C 180,E1 -31091.546,E2 -31091.546} C_VEL
LIN {X 0,Y 26.485,Z 605.738,A -85,B 0,C 180,E1 -31118.255,E2 -31118.255} C_VEL
LIN {X 0,Y 38.932,Z 599.309,A -85,B 0,C 180,E1 -31128.78,E2 -31128.78} C_VEL
LIN {X 0,Y 51.23,Z 591.811,A -85,B 0,C 180,E1 -31134.053,E2 -31134.053} C_VEL
LIN {X 0,Y 63.328,Z 583.055,A -85,B 0,C 180,E1 -31137.215,E2 -31137.215} C_VEL
LIN {X 0,Y 75.555,Z 572.45,A -85,B 0,C 180,E1 -31139.468,E2 -31139.468} C_VEL
LIN {X 0,Y 86.103,Z 561.586,A -85,B 0,C 180,E1 -31140.813,E2 -31140.813} C_VEL
LIN {X 0,Y 95.803,Z 549.733,A -85,B 0,C 180,E1 -31141.78,E2 -31141.78} C_VEL
LIN {X 0,Y 104.643,Z 536.783,A -85,B 0,C 180,E1 -31142.518,E2 -31142.518} C_VEL
LIN {X 0,Y 112.611,Z 522.539,A -85,B 0,C 180,E1 -31143.082,E2 -31143.082} C_VEL
LIN {X 0,Y 119.224,Z 507.769,A -85,B 0,C 180,E1 -31143.464,E2 -31143.464} C_VEL
LIN {X 0,Y 124.07,Z 493.842,A -85,B 0,C 180,E1 -31143.73,E2 -31143.73} C_VEL
LIN {X 0,Y 128.112,Z 477.95,A -85,B 0,C 180,E1 -31143.918,E2 -31143.918} C_VEL
LIN {X 0,Y 131.029,Z 459.697,A -85,B 0,C 180,E1 -31144.179,E2 -31144.179} C_VEL
LIN {X 0,Y 131.119,Z 458.569,A -85,B 0,C 180,E1 -31144.358,E2 -31144.358} C_VEL
LIN {X 0,Y 130.338,Z 454.31,A -85,B 0,C 180,E1 -31148.914,E2 -31148.914} C_VEL
LIN {X 0,Y 130.024,Z 452.357,A -85,B 0,C 180,E1 -31152.481,E2 -31152.481} C_VEL
LIN {X 0,Y 129.916,Z 452.532,A -85,B 0,C 180,E1 -31156.695,E2 -31156.695} C_VEL
LIN {X 0,Y 130.323,Z 455.333,A -85,B 0,C 180,E1 -31162.172,E2 -31162.172} C_VEL
LIN {X 0,Y 130.942,Z 458.165,A -85,B 0,C 180,E1 -31165.534,E2 -31165.534} C_VEL
LIN {X 0,Y 130.94,Z 459.457,A -85,B 0,C 180,E1 -31166.022,E2 -31166.022} C_VEL
LIN {X 0,Y 130.642,Z 461.85,A -85,B 0,C 180,E1 -31166.12,E2 -31166.12} C_VEL
LIN {X 0,Y 129.941,Z 465.483,A -85,B 0,C 180,E1 -31165.637,E2 -31165.637} C_VEL
LIN {X 0,Y 127.908,Z 473.756,A -85,B 0,C 180,E1 -31163.599,E2 -31163.599} C_VEL
LIN {X 0,Y 126.989,Z 477.612,A -85,B 0,C 180,E1 -31163.214,E2 -31163.214} C_VEL
LIN {X 0,Y 126.824,Z 478.406,A -85,B 0,C 180,E1 -31163.222,E2 -31163.222} C_VEL
LIN {X 0,Y 122.795,Z 493.816,A -85,B 0,C 180,E1 -31163.432,E2 -31163.432} C_VEL
LIN {X 0,Y 117.483,Z 508.621,A -85,B 0,C 180,E1 -31163.65,E2 -31163.65} C_VEL
LIN {X 0,Y 110.625,Z 523.507,A -85,B 0,C 180,E1 -31164.042,E2 -31164.042} C_VEL
LIN {X 0,Y 102.65,Z 537.348,A -85,B 0,C 180,E1 -31164.449,E2 -31164.449} C_VEL
LIN {X 0,Y 93.991,Z 549.734,A -85,B 0,C 180,E1 -31164.956,E2 -31164.956} C_VEL
LIN {X 0,Y 84.164,Z 561.519,A -85,B 0,C 180,E1 -31165.639,E2 -31165.639} C_VEL
LIN {X 0,Y 72.73,Z 573.01,A -85,B 0,C 180,E1 -31166.638,E2 -31166.638} C_VEL
LIN {X 0,Y 61.51,Z 582.46,A -85,B 0,C 180,E1 -31167.939,E2 -31167.939} C_VEL
LIN {X 0,Y 48.647,Z 591.52,A -85,B 0,C 180,E1 -31169.905,E2 -31169.905} C_VEL
LIN {X 0,Y 37.211,Z 598.255,A -85,B 0,C 180,E1 -31172.667,E2 -31172.667} C_VEL
LIN {X 0,Y 24.045,Z 604.698,A -85,B 0,C 180,E1 -31178.637,E2 -31178.637} C_VEL
LIN {X 0,Y 11.837,Z 609.616,A -85,B 0,C 180,E1 -31193.56,E2 -31193.56} C_VEL
LIN {X 0,Y 5.052,Z 613.098,A -85,B 0,C 180,E1 -31274.022,E2 -31274.022} C_VEL
LIN {X 0,Y 14.346,Z 615.805,A -85,B 0,C 180,E1 -31331.597,E2 -31331.597} C_VEL
LIN {X 0,Y 14.701,Z 615.904,A -85,B 0,C 180,E1 -31337.071,E2 -31337.071} C_VEL
LIN {X 0,Y 8.768,Z 614.669,A -85,B 0,C 180,E1 -31356.757,E2 -31356.757} C_VEL
LIN {X 0,Y 5.826,Z 613.139,A -85,B 0,C 180,E1 -31410.028,E2 -31410.028} C_VEL
LIN {X 0,Y 11.562,Z 610.134,A -85,B 0,C 180,E1 -31475.779,E2 -31475.779} C_VEL
LIN {X 0,Y 24.742,Z 604.801,A -85,B 0,C 180,E1 -31493.859,E2 -31493.859} C_VEL
LIN {X 0,Y 38.906,Z 597.806,A -85,B 0,C 180,E1 -31499.596,E2 -31499.596} C_VEL
LIN {X 0,Y 52.756,Z 589.334,A -85,B 0,C 180,E1 -31502.339,E2 -31502.339} C_VEL
LIN {X 0,Y 65.164,Z 580.097,A -85,B 0,C 180,E1 -31503.931,E2 -31503.931} C_VEL
LIN {X 0,Y 75.831,Z 570.625,A -85,B 0,C 180,E1 -31504.913,E2 -31504.913} C_VEL
LIN {X 0,Y 86.501,Z 559.467,A -85,B 0,C 180,E1 -31505.561,E2 -31505.561} C_VEL
LIN {X 0,Y 96.294,Z 547.24,A -85,B 0,C 180,E1 -31506.051,E2 -31506.051} C_VEL
LIN {X 0,Y 104.312,Z 535.259,A -85,B 0,C 180,E1 -31506.392,E2 -31506.392} C_VEL
LIN {X 0,Y 111.445,Z 522.477,A -85,B 0,C 180,E1 -31506.666,E2 -31506.666} C_VEL
LIN {X 0,Y 118.139,Z 507.645,A -85,B 0,C 180,E1 -31506.848,E2 -31506.848} C_VEL
LIN {X 0,Y 123.015,Z 493.734,A -85,B 0,C 180,E1 -31506.979,E2 -31506.979} C_VEL
LIN {X 0,Y 127.083,Z 477.825,A -85,B 0,C 180,E1 -31507.072,E2 -31507.072} C_VEL
LIN {X 0,Y 129.504,Z 463.283,A -85,B 0,C 180,E1 -31507.293,E2 -31507.293} C_VEL
LIN {X 0,Y 129.12,Z 460.354,A -85,B 0,C 180,E1 -31510.79,E2 -31510.79} C_VEL
LIN {X 0,Y 129.034,Z 459.375,A -85,B 0,C 180,E1 -31512.578,E2 -31512.578} C_VEL
LIN {X 0,Y 128.936,Z 459.438,A -85,B 0,C 180,E1 -31516.063,E2 -31516.063} C_VEL
LIN {X 0,Y 129.192,Z 462.213,A -85,B 0,C 180,E1 -31521.486,E2 -31521.486} C_VEL
LIN {X 0,Y 129.419,Z 463.33,A -85,B 0,C 180,E1 -31522.988,E2 -31522.988} C_VEL
LIN {X 0,Y 128.095,Z 472.068,A -85,B 0,C 180,E1 -31523.179,E2 -31523.179} C_VEL
LIN {X 0,Y 126.824,Z 478.406,A -85,B 0,C 180,E1 -31523.222,E2 -31523.222} C_VEL
LIN {X 0,Y 125.468,Z 484.136,A -85,B 0,C 180,E1 -31523.063,E2 -31523.063} C_VEL
LIN {X 0,Y 122.611,Z 493.265,A -85,B 0,C 180,E1 -31521.836,E2 -31521.836} C_VEL
LIN {X 0,Y 119.303,Z 502.237,A -85,B 0,C 180,E1 -31520.473,E2 -31520.473} C_VEL
LIN {X 0,Y 117.872,Z 505.894,A -85,B 0,C 180,E1 -31520.208,E2 -31520.208} C_VEL
LIN {X 0,Y 117.126,Z 507.734,A -85,B 0,C 180,E1 -31520.203,E2 -31520.203} C_VEL
LIN {X 0,Y 110.582,Z 522.154,A -85,B 0,C 180,E1 -31520.375,E2 -31520.375} C_VEL
LIN {X 0,Y 102.941,Z 535.692,A -85,B 0,C 180,E1 -31520.498,E2 -31520.498} C_VEL
LIN {X 0,Y 93.871,Z 548.894,A -85,B 0,C 180,E1 -31520.631,E2 -31520.631} C_VEL
LIN {X 0,Y 83.652,Z 561.229,A -85,B 0,C 180,E1 -31520.825,E2 -31520.825} C_VEL
LIN {X 0,Y 73.412,Z 571.617,A -85,B 0,C 180,E1 -31521.025,E2 -31521.025} C_VEL
LIN {X 0,Y 62.234,Z 581.224,A -85,B 0,C 180,E1 -31521.302,E2 -31521.302} C_VEL
LIN {X 0,Y 49.105,Z 590.619,A -85,B 0,C 180,E1 -31521.514,E2 -31521.514} C_VEL
LIN {X 0,Y 37.813,Z 597.391,A -85,B 0,C 180,E1 -31521.664,E2 -31521.664} C_VEL
LIN {X 0,Y 26.457,Z 603.041,A -85,B 0,C 180,E1 -31521.593,E2 -31521.593} C_VEL
LIN {X 0,Y 14.961,Z 607.796,A -85,B 0,C 180,E1 -31520.002,E2 -31520.002} C_VEL
LIN {X 0,Y 12.508,Z 608.675,A -85,B 0,C 180,E1 -31518.674,E2 -31518.674} C_VEL
LIN {X 0,Y 14.353,Z 608.058,A -85,B 0,C 180,E1 -31511.626,E2 -31511.626} C_VEL
LIN {X 0,Y 28.569,Z 602.171,A -85,B 0,C 180,E1 -31510.239,E2 -31510.239} C_VEL
LIN {X 0,Y 42.832,Z 594.673,A -85,B 0,C 180,E1 -31510.084,E2 -31510.084} C_VEL
LIN {X 0,Y 55.32,Z 586.604,A -85,B 0,C 180,E1 -31510.065,E2 -31510.065} C_VEL
LIN {X 0,Y 67.849,Z 576.831,A -85,B 0,C 180,E1 -31510.246,E2 -31510.246} C_VEL
LIN {X 0,Y 78.924,Z 566.501,A -85,B 0,C 180,E1 -31510.25,E2 -31510.25} C_VEL
LIN {X 0,Y 89.284,Z 554.999,A -85,B 0,C 180,E1 -31510.28,E2 -31510.28} C_VEL
LIN {X 0,Y 99.108,Z 541.9,A -85,B 0,C 180,E1 -31510.289,E2 -31510.289} C_VEL
LIN {X 0,Y 107.148,Z 528.905,A -85,B 0,C 180,E1 -31510.304,E2 -31510.304} C_VEL
LIN {X 0,Y 114.3,Z 514.722,A -85,B 0,C 180,E1 -31510.327,E2 -31510.327} C_VEL
LIN {X 0,Y 120.111,Z 500.183,A -85,B 0,C 180,E1 -31510.237,E2 -31510.237} C_VEL
LIN {X 0,Y 124.746,Z 484.671,A -85,B 0,C 180,E1 -31510.25,E2 -31510.25} C_VEL
LIN {X 0,Y 127.925,Z 469.02,A -85,B 0,C 180,E1 -31510.304,E2 -31510.304} C_VEL
LIN {X 0,Y 128.078,Z 468.036,A -85,B 0,C 180,E1 -31510.347,E2 -31510.347} C_VEL
LIN {X 0,Y 128.013,Z 466.551,A -85,B 0,C 180,E1 -31512.68,E2 -31512.68} C_VEL
LIN {X 0,Y 127.902,Z 466.727,A -85,B 0,C 180,E1 -31516.197,E2 -31516.197} C_VEL
LIN {X 0,Y 127.96,Z 468.409,A -85,B 0,C 180,E1 -31519.937,E2 -31519.937} C_VEL
LIN {X 0,Y 125.045,Z 483.073,A -85,B 0,C 180,E1 -31520.048,E2 -31520.048} C_VEL
LIN {X 0,Y 120.614,Z 498.349,A -85,B 0,C 180,E1 -31520.175,E2 -31520.175} C_VEL
LIN {X 0,Y 117.126,Z 507.734,A -85,B 0,C 180,E1 -31520.203,E2 -31520.203} C_VEL
LIN {X 0,Y 114.826,Z 513.17,A -85,B 0,C 180,E1 -31519.93,E2 -31519.93} C_VEL
LIN {X 0,Y 110.661,Z 521.717,A -85,B 0,C 180,E1 -31518.527,E2 -31518.527} C_VEL
LIN {X 0,Y 106.089,Z 530.06,A -85,B 0,C 180,E1 -31516.98,E2 -31516.98} C_VEL
LIN {X 0,Y 103.073,Z 535.078,A -85,B 0,C 180,E1 -31516.551,E2 -31516.551} C_VEL
LIN {X 0,Y 94.286,Z 548.052,A -85,B 0,C 180,E1 -31516.321,E2 -31516.321} C_VEL
LIN {X 0,Y 84.073,Z 560.56,A -85,B 0,C 180,E1 -31515.984,E2 -31515.984} C_VEL
LIN {X 0,Y 77.803,Z 567.214,A -85,B 0,C 180,E1 -31515.714,E2 -31515.714} C_VEL
LIN {X 0,Y 80.16,Z 564.819,A -85,B 0,C 180,E1 -31515.327,E2 -31515.327} C_VEL
LIN {X 0,Y 89.952,Z 553.68,A -85,B 0,C 180,E1 -31514.789,E2 -31514.789} C_VEL
LIN {X 0,Y 98.919,Z 541.567,A -85,B 0,C 180,E1 -31514.389,E2 -31514.389} C_VEL
LIN {X 0,Y 106.881,Z 528.653,A -85,B 0,C 180,E1 -31514.093,E2 -31514.093} C_VEL
LIN {X 0,Y 114.017,Z 514.465,A -85,B 0,C 180,E1 -31513.872,E2 -31513.872} C_VEL
LIN {X 0,Y 119.995,Z 499.369,A -85,B 0,C 180,E1 -31513.606,E2 -31513.606} C_VEL
LIN {X 0,Y 124.459,Z 484.27,A -85,B 0,C 180,E1 -31513.513,E2 -31513.513} C_VEL
LIN {X 0,Y 126.812,Z 473.562,A -85,B 0,C 180,E1 -31513.502,E2 -31513.502} C_VEL
LIN {X 0,Y 126.734,Z 473.807,A -85,B 0,C 180,E1 -31516.092,E2 -31516.092} C_VEL
LIN {X 0,Y 126.675,Z 474.172,A -85,B 0,C 180,E1 -31516.822,E2 -31516.822} C_VEL
LIN {X 0,Y 122.979,Z 489.817,A -85,B 0,C 180,E1 -31516.798,E2 -31516.798} C_VEL
LIN {X 0,Y 117.945,Z 504.968,A -85,B 0,C 180,E1 -31516.749,E2 -31516.749} C_VEL
LIN {X 0,Y 111.897,Z 519.003,A -85,B 0,C 180,E1 -31516.7,E2 -31516.7} C_VEL
LIN {X 0,Y 104.494,Z 532.784,A -85,B 0,C 180,E1 -31516.579,E2 -31516.579} C_VEL
LIN {X 0,Y 103.073,Z 535.078,A -85,B 0,C 180,E1 -31516.551,E2 -31516.551} C_VEL
LIN {X 0,Y 102.773,Z 536.132,A -85,B 0,C 180,E1 -31516.543,E2 -31516.543} C_VEL
LIN {X 0,Y 102.773,Z 600,A -85,B 0,C 180,E1 -31516.543,E2 -31516.543} C_VEL
LIN {X 0,Y 102.773,Z 600,A -85,B 0,C 180,E1 -31516.543,E2 -31516.543}

QRS_NEXT_CUT()

QRS_NEXT()
QRS_HOME()

END
